LIN {X 0,Y 572.962,Z 472.956,A -85,B 0,C 180,E1 -2254.924,E2 -2254.924} C_VEL
LIN {X 0,Y 573.098,Z 467.876,A -85,B 0,C 180,E1 -2255.981,E2 -2255.981} C_VEL
LIN {X 0,Y 573.102,Z 461.481,A -85,B 0,C 180,E1 -2257.042,E2 -2257.042} C_VEL
LIN {X 0,Y 573.176,Z 453.495,A -85,B 0,C 180,E1 -2258.104,E2 -2258.104} C_VEL
LIN {X 0,Y 573.253,Z 445.356,A -85,B 0,C 180,E1 -2258.991,E2 -2258.991} C_VEL
LIN {X 0,Y 573.348,Z 435.426,A -85,B 0,C 180,E1 -2259.879,E2 -2259.879} C_VEL
LIN {X 0,Y 573.504,Z 424.221,A -85,B 0,C 180,E1 -2260.679,E2 -2260.679} C_VEL
LIN {X 0,Y 573.624,Z 413.221,A -85,B 0,C 180,E1 -2261.303,E2 -2261.303} C_VEL
LIN {X 0,Y 573.702,Z 401.041,A -85,B 0,C 180,E1 -2261.838,E2 -2261.838} C_VEL
LIN {X 0,Y 573.81,Z 388.273,A -85,B 0,C 180,E1 -2262.24,E2 -2262.24} C_VEL
LIN {X 0,Y 573.89,Z 374.763,A -85,B 0,C 180,E1 -2262.507,E2 -2262.507} C_VEL
LIN {X 0,Y 573.929,Z 274.251,A -85,B 0,C 180,E1 -2263.776,E2 -2263.776} C_VEL
LIN {X 0,Y 573.424,Z 270.457,A -85,B 0,C 180,E1 -2263.847,E2 -2263.847} C_VEL
LIN {X 0,Y 573.615,Z 247.392,A -85,B 0,C 180,E1 -2267.001,E2 -2267.001} C_VEL
LIN {X 0,Y 573.874,Z 225.362,A -85,B 0,C 180,E1 -2270.051,E2 -2270.051} C_VEL
LIN {X 0,Y 574.038,Z 204.991,A -85,B 0,C 180,E1 -2272.871,E2 -2272.871} C_VEL
LIN {X 0,Y 573.669,Z 200.428,A -85,B 0,C 180,E1 -2273.527,E2 -2273.527} C_VEL
LIN {X 0,Y 573.234,Z 198.084,A -85,B 0,C 180,E1 -2273.91,E2 -2273.91} C_VEL
LIN {X 0,Y 573.256,Z 198.078,A -85,B 0,C 180,E1 -2276.496,E2 -2276.496} C_VEL
LIN {X 0,Y 573.25,Z 198.075,A -85,B 0,C 180,E1 -2279.362,E2 -2279.362} C_VEL
LIN {X 0,Y 573.232,Z 198.082,A -85,B 0,C 180,E1 -2282.225,E2 -2282.225} C_VEL
LIN {X 0,Y 573.229,Z 198.076,A -85,B 0,C 180,E1 -2284.77,E2 -2284.77} C_VEL
LIN {X 0,Y 573.23,Z 198.076,A -85,B 0,C 180,E1 -2287.162,E2 -2287.162} C_VEL
LIN {X 0,Y 573.223,Z 198.081,A -85,B 0,C 180,E1 -2289.603,E2 -2289.603} C_VEL
LIN {X 0,Y 573.213,Z 198.078,A -85,B 0,C 180,E1 -2292.638,E2 -2292.638} C_VEL
LIN {X 0,Y 573.206,Z 198.085,A -85,B 0,C 180,E1 -2295.663,E2 -2295.663} C_VEL
LIN {X 0,Y 573.225,Z 198.076,A -85,B 0,C 180,E1 -2298.542,E2 -2298.542} C_VEL
LIN {X 0,Y 573.214,Z 198.08,A -85,B 0,C 180,E1 -2301.296,E2 -2301.296} C_VEL
LIN {X 0,Y 573.224,Z 198.081,A -85,B 0,C 180,E1 -2304.008,E2 -2304.008} C_VEL
LIN {X 0,Y 573.241,Z 198.074,A -85,B 0,C 180,E1 -2306.516,E2 -2306.516} C_VEL
LIN {X 0,Y 573.202,Z 198.081,A -85,B 0,C 180,E1 -2309.111,E2 -2309.111} C_VEL
LIN {X 0,Y 573.23,Z 198.083,A -85,B 0,C 180,E1 -2311.435,E2 -2311.435} C_VEL
LIN {X 0,Y 573.242,Z 198.079,A -85,B 0,C 180,E1 -2313.809,E2 -2313.809} C_VEL
LIN {X 0,Y 573.254,Z 198.074,A -85,B 0,C 180,E1 -2316.901,E2 -2316.901} C_VEL
LIN {X 0,Y 573.216,Z 198.079,A -85,B 0,C 180,E1 -2319.922,E2 -2319.922} C_VEL
LIN {X 0,Y 573.234,Z 198.079,A -85,B 0,C 180,E1 -2322.978,E2 -2322.978} C_VEL
LIN {X 0,Y 573.226,Z 198.078,A -85,B 0,C 180,E1 -2325.806,E2 -2325.806} C_VEL
LIN {X 0,Y 573.277,Z 198.071,A -85,B 0,C 180,E1 -2328.706,E2 -2328.706} C_VEL
LIN {X 0,Y 573.254,Z 198.077,A -85,B 0,C 180,E1 -2331.54,E2 -2331.54} C_VEL
LIN {X 0,Y 573.202,Z 198.082,A -85,B 0,C 180,E1 -2333.664,E2 -2333.664} C_VEL
LIN {X 0,Y 573.174,Z 198.084,A -85,B 0,C 180,E1 -2335.781,E2 -2335.781} C_VEL
LIN {X 0,Y 573.247,Z 198.074,A -85,B 0,C 180,E1 -2337.892,E2 -2337.892} C_VEL
LIN {X 0,Y 573.287,Z 198.072,A -85,B 0,C 180,E1 -2340.702,E2 -2340.702} C_VEL
LIN {X 0,Y 573.196,Z 198.082,A -85,B 0,C 180,E1 -2343.515,E2 -2343.515} C_VEL
LIN {X 0,Y 573.239,Z 198.075,A -85,B 0,C 180,E1 -2345.628,E2 -2345.628} C_VEL
LIN {X 0,Y 573.248,Z 198.076,A -85,B 0,C 180,E1 -2348.46,E2 -2348.46} C_VEL
LIN {X 0,Y 573.266,Z 198.074,A -85,B 0,C 180,E1 -2351.312,E2 -2351.312} C_VEL
LIN {X 0,Y 573.221,Z 198.08,A -85,B 0,C 180,E1 -2354.426,E2 -2354.426} C_VEL
LIN {X 0,Y 573.245,Z 198.078,A -85,B 0,C 180,E1 -2357.112,E2 -2357.112} C_VEL
LIN {X 0,Y 573.21,Z 198.079,A -85,B 0,C 180,E1 -2360.078,E2 -2360.078} C_VEL
LIN {X 0,Y 573.218,Z 198.08,A -85,B 0,C 180,E1 -2363.156,E2 -2363.156} C_VEL
LIN {X 0,Y 573.202,Z 198.085,A -85,B 0,C 180,E1 -2364.418,E2 -2364.418} C_VEL
LIN {X 0,Y 572.571,Z 198.169,A -85,B 0,C 180,E1 -2365.004,E2 -2365.004} C_VEL
LIN {X 0,Y 569.731,Z 198.522,A -85,B 0,C 180,E1 -2365.956,E2 -2365.956} C_VEL
LIN {X 0,Y 567.305,Z 198.822,A -85,B 0,C 180,E1 -2366.722,E2 -2366.722} C_VEL
LIN {X 0,Y 566.255,Z 198.945,A -85,B 0,C 180,E1 -2367.314,E2 -2367.314} C_VEL
LIN {X 0,Y 566.166,Z 198.955,A -85,B 0,C 180,E1 -2367.514,E2 -2367.514} C_VEL
LIN {X 0,Y 566.154,Z 198.957,A -85,B 0,C 180,E1 -2369.771,E2 -2369.771} C_VEL
LIN {X 0,Y 566.165,Z 198.964,A -85,B 0,C 180,E1 -2372.434,E2 -2372.434} C_VEL
LIN {X 0,Y 566.169,Z 198.957,A -85,B 0,C 180,E1 -2374.997,E2 -2374.997} C_VEL
LIN {X 0,Y 566.154,Z 198.957,A -85,B 0,C 180,E1 -2377.464,E2 -2377.464} C_VEL
LIN {X 0,Y 566.185,Z 198.96,A -85,B 0,C 180,E1 -2380.201,E2 -2380.201} C_VEL
LIN {X 0,Y 566.173,Z 198.955,A -85,B 0,C 180,E1 -2383.057,E2 -2383.057} C_VEL
LIN {X 0,Y 566.163,Z 198.962,A -85,B 0,C 180,E1 -2386.052,E2 -2386.052} C_VEL
LIN {X 0,Y 566.181,Z 198.955,A -85,B 0,C 180,E1 -2388.867,E2 -2388.867} C_VEL
LIN {X 0,Y 566.158,Z 198.958,A -85,B 0,C 180,E1 -2391.64,E2 -2391.64} C_VEL
LIN {X 0,Y 566.179,Z 198.961,A -85,B 0,C 180,E1 -2394.314,E2 -2394.314} C_VEL
LIN {X 0,Y 566.205,Z 198.951,A -85,B 0,C 180,E1 -2396.902,E2 -2396.902} C_VEL
LIN {X 0,Y 566.164,Z 198.957,A -85,B 0,C 180,E1 -2399.411,E2 -2399.411} C_VEL
LIN {X 0,Y 566.194,Z 198.959,A -85,B 0,C 180,E1 -2401.861,E2 -2401.861} C_VEL
LIN {X 0,Y 566.199,Z 198.956,A -85,B 0,C 180,E1 -2404.254,E2 -2404.254} C_VEL
LIN {X 0,Y 566.156,Z 198.957,A -85,B 0,C 180,E1 -2406.722,E2 -2406.722} C_VEL
LIN {X 0,Y 566.193,Z 198.958,A -85,B 0,C 180,E1 -2409.665,E2 -2409.665} C_VEL
LIN {X 0,Y 566.179,Z 198.954,A -85,B 0,C 180,E1 -2412.671,E2 -2412.671} C_VEL
LIN {X 0,Y 566.213,Z 198.957,A -85,B 0,C 180,E1 -2415.629,E2 -2415.629} C_VEL
LIN {X 0,Y 566.23,Z 198.947,A -85,B 0,C 180,E1 -2418.678,E2 -2418.678} C_VEL
LIN {X 0,Y 566.219,Z 198.954,A -85,B 0,C 180,E1 -2421.436,E2 -2421.436} C_VEL
LIN {X 0,Y 566.249,Z 198.948,A -85,B 0,C 180,E1 -2424.303,E2 -2424.303} C_VEL
LIN {X 0,Y 566.2,Z 199.072,A -85,B 0,C 180,E1 -2426.621,E2 -2426.621} C_VEL
LIN {X 0,Y 566.394,Z 207.555,A -85,B 0,C 180,E1 -2428.224,E2 -2428.224} C_VEL
LIN {X 0,Y 566.201,Z 222.6,A -85,B 0,C 180,E1 -2431.046,E2 -2431.046} C_VEL
LIN {X 0,Y 567.188,Z 228.36,A -85,B 0,C 180,E1 -2431.155,E2 -2431.155} C_VEL
LIN {X 0,Y 566.924,Z 328.742,A -85,B 0,C 180,E1 -2432.443,E2 -2432.443} C_VEL
LIN {X 0,Y 566.819,Z 341.931,A -85,B 0,C 180,E1 -2432.755,E2 -2432.755} C_VEL
LIN {X 0,Y 566.731,Z 354.545,A -85,B 0,C 180,E1 -2433.2,E2 -2433.2} C_VEL
LIN {X 0,Y 566.593,Z 365.826,A -85,B 0,C 180,E1 -2433.735,E2 -2433.735} C_VEL
LIN {X 0,Y 566.423,Z 377.466,A -85,B 0,C 180,E1 -2434.448,E2 -2434.448} C_VEL
LIN {X 0,Y 566.31,Z 387.918,A -85,B 0,C 180,E1 -2435.252,E2 -2435.252} C_VEL
LIN {X 0,Y 566.171,Z 396.509,A -85,B 0,C 180,E1 -2436.057,E2 -2436.057} C_VEL
LIN {X 0,Y 566.112,Z 404.244,A -85,B 0,C 180,E1 -2436.93,E2 -2436.93} C_VEL
LIN {X 0,Y 566.044,Z 412.234,A -85,B 0,C 180,E1 -2438.03,E2 -2438.03} C_VEL
LIN {X 0,Y 565.982,Z 417.564,A -85,B 0,C 180,E1 -2438.93,E2 -2438.93} C_VEL
LIN {X 0,Y 565.946,Z 422.761,A -85,B 0,C 180,E1 -2440.012,E2 -2440.012} C_VEL
LIN {X 0,Y 565.91,Z 426.988,A -85,B 0,C 180,E1 -2441.159,E2 -2441.159} C_VEL
LIN {X 0,Y 565.868,Z 429.791,A -85,B 0,C 180,E1 -2442.189,E2 -2442.189} C_VEL
LIN {X 0,Y 565.844,Z 431.212,A -85,B 0,C 180,E1 -2442.919,E2 -2442.919} C_VEL
LIN {X 0,Y 565.862,Z 432.216,A -85,B 0,C 180,E1 -2443.649,E2 -2443.649} C_VEL
LIN {X 0,Y 565.875,Z 432.818,A -85,B 0,C 180,E1 -2444.382,E2 -2444.382} C_VEL
LIN {X 0,Y 565.803,Z 432.99,A -85,B 0,C 180,E1 -2445.12,E2 -2445.12} C_VEL
LIN {X 0,Y 565.81,Z 432.718,A -85,B 0,C 180,E1 -2445.858,E2 -2445.858} C_VEL
LIN {X 0,Y 565.852,Z 431.495,A -85,B 0,C 180,E1 -2446.991,E2 -2446.991} C_VEL
LIN {X 0,Y 565.892,Z 428.378,A -85,B 0,C 180,E1 -2448.463,E2 -2448.463} C_VEL
LIN {X 0,Y 565.927,Z 424.709,A -85,B 0,C 180,E1 -2449.59,E2 -2449.59} C_VEL
LIN {X 0,Y 565.945,Z 419.781,A -85,B 0,C 180,E1 -2450.726,E2 -2450.726} C_VEL
LIN {X 0,Y 566.005,Z 413.426,A -85,B 0,C 180,E1 -2451.869,E2 -2451.869} C_VEL
LIN {X 0,Y 566.078,Z 405.548,A -85,B 0,C 180,E1 -2452.998,E2 -2452.998} C_VEL
LIN {X 0,Y 566.185,Z 396.971,A -85,B 0,C 180,E1 -2453.986,E2 -2453.986} C_VEL
LIN {X 0,Y 566.313,Z 386.516,A -85,B 0,C 180,E1 -2454.956,E2 -2454.956} C_VEL
LIN {X 0,Y 566.431,Z 376.094,A -85,B 0,C 180,E1 -2455.737,E2 -2455.737} C_VEL
LIN {X 0,Y 566.607,Z 364.554,A -85,B 0,C 180,E1 -2456.421,E2 -2456.421} C_VEL
LIN {X 0,Y 566.73,Z 351.798,A -85,B 0,C 180,E1 -2457.001,E2 -2457.001} C_VEL
LIN {X 0,Y 566.834,Z 339.084,A -85,B 0,C 180,E1 -2457.418,E2 -2457.418} C_VEL
LIN {X 0,Y 566.894,Z 326.866,A -85,B 0,C 180,E1 -2457.677,E2 -2457.677} C_VEL
LIN {X 0,Y 567.16,Z 228.196,A -85,B 0,C 180,E1 -2458.938,E2 -2458.938} C_VEL
LIN {X 0,Y 566.194,Z 222.551,A -85,B 0,C 180,E1 -2459.053,E2 -2459.053} C_VEL
LIN {X 0,Y 566.348,Z 207.789,A -85,B 0,C 180,E1 -2461.828,E2 -2461.828} C_VEL
LIN {X 0,Y 566.256,Z 198.949,A -85,B 0,C 180,E1 -2463.465,E2 -2463.465} C_VEL
LIN {X 0,Y 566.205,Z 198.959,A -85,B 0,C 180,E1 -2466.567,E2 -2466.567} C_VEL
LIN {X 0,Y 566.201,Z 198.953,A -85,B 0,C 180,E1 -2469.684,E2 -2469.684} C_VEL
LIN {X 0,Y 566.214,Z 198.956,A -85,B 0,C 180,E1 -2472.084,E2 -2472.084} C_VEL
LIN {X 0,Y 566.156,Z 198.958,A -85,B 0,C 180,E1 -2475.034,E2 -2475.034} C_VEL
LIN {X 0,Y 566.206,Z 198.956,A -85,B 0,C 180,E1 -2477.912,E2 -2477.912} C_VEL
LIN {X 0,Y 566.204,Z 198.953,A -85,B 0,C 180,E1 -2480.726,E2 -2480.726} C_VEL
LIN {X 0,Y 566.195,Z 198.957,A -85,B 0,C 180,E1 -2483.782,E2 -2483.782} C_VEL
LIN {X 0,Y 566.205,Z 198.956,A -85,B 0,C 180,E1 -2486.261,E2 -2486.261} C_VEL
LIN {X 0,Y 566.179,Z 198.953,A -85,B 0,C 180,E1 -2488.919,E2 -2488.919} C_VEL
LIN {X 0,Y 566.2,Z 198.959,A -85,B 0,C 180,E1 -2491.791,E2 -2491.791} C_VEL
LIN {X 0,Y 566.197,Z 198.954,A -85,B 0,C 180,E1 -2494.25,E2 -2494.25} C_VEL
LIN {X 0,Y 566.207,Z 198.95,A -85,B 0,C 180,E1 -2496.701,E2 -2496.701} C_VEL
LIN {X 0,Y 566.195,Z 198.96,A -85,B 0,C 180,E1 -2499.662,E2 -2499.662} C_VEL
LIN {X 0,Y 566.242,Z 198.946,A -85,B 0,C 180,E1 -2502.868,E2 -2502.868} C_VEL
LIN {X 0,Y 566.207,Z 198.959,A -85,B 0,C 180,E1 -2505.626,E2 -2505.626} C_VEL
LIN {X 0,Y 566.24,Z 198.946,A -85,B 0,C 180,E1 -2508.653,E2 -2508.653} C_VEL
LIN {X 0,Y 566.217,Z 198.957,A -85,B 0,C 180,E1 -2511.434,E2 -2511.434} C_VEL
LIN {X 0,Y 566.186,Z 198.959,A -85,B 0,C 180,E1 -2513.586,E2 -2513.586} C_VEL
LIN {X 0,Y 566.154,Z 198.959,A -85,B 0,C 180,E1 -2515.729,E2 -2515.729} C_VEL
LIN {X 0,Y 566.239,Z 198.948,A -85,B 0,C 180,E1 -2517.866,E2 -2517.866} C_VEL
LIN {X 0,Y 566.244,Z 198.945,A -85,B 0,C 180,E1 -2520,E2 -2520} C_VEL
LIN {X 0,Y 566.243,Z 198.949,A -85,B 0,C 180,E1 -2522.846,E2 -2522.846} C_VEL
LIN {X 0,Y 566.225,Z 198.948,A -85,B 0,C 180,E1 -2525.699,E2 -2525.699} C_VEL
LIN {X 0,Y 566.17,Z 198.957,A -85,B 0,C 180,E1 -2528.567,E2 -2528.567} C_VEL
LIN {X 0,Y 566.226,Z 198.95,A -85,B 0,C 180,E1 -2531.455,E2 -2531.455} C_VEL
LIN {X 0,Y 566.192,Z 198.954,A -85,B 0,C 180,E1 -2534.505,E2 -2534.505} C_VEL
LIN {X 0,Y 566.162,Z 198.958,A -85,B 0,C 180,E1 -2537.333,E2 -2537.333} C_VEL
LIN {X 0,Y 566.178,Z 198.956,A -85,B 0,C 180,E1 -2540.339,E2 -2540.339} C_VEL
LIN {X 0,Y 566.133,Z 198.961,A -85,B 0,C 180,E1 -2543.281,E2 -2543.281} C_VEL
LIN {X 0,Y 566.167,Z 198.955,A -85,B 0,C 180,E1 -2545.752,E2 -2545.752} C_VEL
LIN {X 0,Y 566.156,Z 198.959,A -85,B 0,C 180,E1 -2548.2,E2 -2548.2} C_VEL
LIN {X 0,Y 566.159,Z 198.958,A -85,B 0,C 180,E1 -2551.077,E2 -2551.077} C_VEL
LIN {X 0,Y 566.171,Z 198.955,A -85,B 0,C 180,E1 -2553.734,E2 -2553.734} C_VEL
LIN {X 0,Y 566.159,Z 198.964,A -85,B 0,C 180,E1 -2556.573,E2 -2556.573} C_VEL
LIN {X 0,Y 566.191,Z 198.954,A -85,B 0,C 180,E1 -2559.687,E2 -2559.687} C_VEL
LIN {X 0,Y 566.193,Z 198.956,A -85,B 0,C 180,E1 -2562.09,E2 -2562.09} C_VEL
LIN {X 0,Y 566.152,Z 198.958,A -85,B 0,C 180,E1 -2565.038,E2 -2565.038} C_VEL
LIN {X 0,Y 566.162,Z 198.961,A -85,B 0,C 180,E1 -2567.911,E2 -2567.911} C_VEL
LIN {X 0,Y 566.199,Z 198.953,A -85,B 0,C 180,E1 -2570.728,E2 -2570.728} C_VEL
LIN {X 0,Y 566.193,Z 198.957,A -85,B 0,C 180,E1 -2573.787,E2 -2573.787} C_VEL
LIN {X 0,Y 566.204,Z 198.957,A -85,B 0,C 180,E1 -2576.268,E2 -2576.268} C_VEL
LIN {X 0,Y 566.183,Z 198.954,A -85,B 0,C 180,E1 -2578.926,E2 -2578.926} C_VEL
LIN {X 0,Y 566.184,Z 198.963,A -85,B 0,C 180,E1 -2581.857,E2 -2581.857} C_VEL
LIN {X 0,Y 566.204,Z 198.957,A -85,B 0,C 180,E1 -2584.252,E2 -2584.252} C_VEL
LIN {X 0,Y 566.222,Z 199.029,A -85,B 0,C 180,E1 -2586.016,E2 -2586.016} C_VEL
LIN {X 0,Y 567.041,Z 204.539,A -85,B 0,C 180,E1 -2586.828,E2 -2586.828} C_VEL
LIN {X 0,Y 566.895,Z 223.622,A -85,B 0,C 180,E1 -2589.5,E2 -2589.5} C_VEL
LIN {X 0,Y 566.663,Z 243.988,A -85,B 0,C 180,E1 -2592.311,E2 -2592.311} C_VEL
LIN {X 0,Y 566.474,Z 265.273,A -85,B 0,C 180,E1 -2595.264,E2 -2595.264} C_VEL
LIN {X 0,Y 566.411,Z 270.522,A -85,B 0,C 180,E1 -2595.987,E2 -2595.987} C_VEL
LIN {X 0,Y 567.165,Z 277.243,A -85,B 0,C 180,E1 -2596.095,E2 -2596.095} C_VEL
LIN {X 0,Y 566.971,Z 378.942,A -85,B 0,C 180,E1 -2597.403,E2 -2597.403} C_VEL
LIN {X 0,Y 566.843,Z 392.214,A -85,B 0,C 180,E1 -2597.719,E2 -2597.719} C_VEL
LIN {X 0,Y 566.741,Z 404.374,A -85,B 0,C 180,E1 -2598.148,E2 -2598.148} C_VEL
LIN {X 0,Y 566.629,Z 416.064,A -85,B 0,C 180,E1 -2598.703,E2 -2598.703} C_VEL
LIN {X 0,Y 566.486,Z 426.902,A -85,B 0,C 180,E1 -2599.365,E2 -2599.365} C_VEL
LIN {X 0,Y 566.337,Z 437.535,A -85,B 0,C 180,E1 -2600.175,E2 -2600.175} C_VEL
LIN {X 0,Y 566.207,Z 447.109,A -85,B 0,C 180,E1 -2601.074,E2 -2601.074} C_VEL
LIN {X 0,Y 566.113,Z 454.956,A -85,B 0,C 180,E1 -2601.971,E2 -2601.971} C_VEL
LIN {X 0,Y 566.002,Z 462.619,A -85,B 0,C 180,E1 -2603.046,E2 -2603.046} C_VEL
LIN {X 0,Y 566.004,Z 469.676,A -85,B 0,C 180,E1 -2604.298,E2 -2604.298} C_VEL
LIN {X 0,Y 565.933,Z 474.369,A -85,B 0,C 180,E1 -2605.369,E2 -2605.369} C_VEL
LIN {X 0,Y 565.927,Z 477.955,A -85,B 0,C 180,E1 -2606.439,E2 -2606.439} C_VEL
LIN {X 0,Y 565.878,Z 479.805,A -85,B 0,C 180,E1 -2607.151,E2 -2607.151} C_VEL
LIN {X 0,Y 565.846,Z 482.183,A -85,B 0,C 180,E1 -2608.575,E2 -2608.575} C_VEL
LIN {X 0,Y 565.839,Z 483,A -85,B 0,C 180,E1 -2609.999,E2 -2609.999} C_VEL
LIN {X 0,Y 565.846,Z 482.187,A -85,B 0,C 180,E1 -2611.422,E2 -2611.422} C_VEL
LIN {X 0,Y 565.877,Z 479.813,A -85,B 0,C 180,E1 -2612.846,E2 -2612.846} C_VEL
LIN {X 0,Y 565.926,Z 476.9,A -85,B 0,C 180,E1 -2613.915,E2 -2613.915} C_VEL
LIN {X 0,Y 565.877,Z 472.955,A -85,B 0,C 180,E1 -2614.986,E2 -2614.986} C_VEL
LIN {X 0,Y 566.007,Z 467.876,A -85,B 0,C 180,E1 -2616.057,E2 -2616.057} C_VEL
LIN {X 0,Y 566.039,Z 461.481,A -85,B 0,C 180,E1 -2617.13,E2 -2617.13} C_VEL
LIN {X 0,Y 566.132,Z 453.494,A -85,B 0,C 180,E1 -2618.206,E2 -2618.206} C_VEL
LIN {X 0,Y 566.227,Z 445.355,A -85,B 0,C 180,E1 -2619.103,E2 -2619.103} C_VEL
LIN {X 0,Y 566.349,Z 435.425,A -85,B 0,C 180,E1 -2620.003,E2 -2620.003} C_VEL
LIN {X 0,Y 566.508,Z 424.32,A -85,B 0,C 180,E1 -2620.806,E2 -2620.806} C_VEL
LIN {X 0,Y 566.656,Z 413.219,A -85,B 0,C 180,E1 -2621.443,E2 -2621.443} C_VEL
LIN {X 0,Y 566.756,Z 401.039,A -85,B 0,C 180,E1 -2621.985,E2 -2621.985} C_VEL
LIN {X 0,Y 566.894,Z 388.272,A -85,B 0,C 180,E1 -2622.391,E2 -2622.391} C_VEL
LIN {X 0,Y 566.971,Z 374.762,A -85,B 0,C 180,E1 -2622.662,E2 -2622.662} C_VEL
LIN {X 0,Y 567.043,Z 274.921,A -85,B 0,C 180,E1 -2623.938,E2 -2623.938} C_VEL
LIN {X 0,Y 566.428,Z 270.457,A -85,B 0,C 180,E1 -2624.022,E2 -2624.022} C_VEL
LIN {X 0,Y 566.642,Z 248.047,A -85,B 0,C 180,E1 -2627.125,E2 -2627.125} C_VEL
LIN {X 0,Y 566.901,Z 226.406,A -85,B 0,C 180,E1 -2630.119,E2 -2630.119} C_VEL
LIN {X 0,Y 567.105,Z 206.052,A -85,B 0,C 180,E1 -2632.974,E2 -2632.974} C_VEL
LIN {X 0,Y 566.796,Z 202.108,A -85,B 0,C 180,E1 -2633.548,E2 -2633.548} C_VEL
LIN {X 0,Y 566.207,Z 198.96,A -85,B 0,C 180,E1 -2634.03,E2 -2634.03} C_VEL
LIN {X 0,Y 566.221,Z 198.953,A -85,B 0,C 180,E1 -2636.661,E2 -2636.661} C_VEL
LIN {X 0,Y 566.188,Z 198.958,A -85,B 0,C 180,E1 -2639.765,E2 -2639.765} C_VEL
LIN {X 0,Y 566.185,Z 198.957,A -85,B 0,C 180,E1 -2642.426,E2 -2642.426} C_VEL
LIN {X 0,Y 566.191,Z 198.952,A -85,B 0,C 180,E1 -2644.991,E2 -2644.991} C_VEL
LIN {X 0,Y 566.173,Z 198.957,A -85,B 0,C 180,E1 -2647.457,E2 -2647.457} C_VEL
LIN {X 0,Y 566.201,Z 198.956,A -85,B 0,C 180,E1 -2650.194,E2 -2650.194} C_VEL
LIN {X 0,Y 566.175,Z 198.954,A -85,B 0,C 180,E1 -2653.05,E2 -2653.05} C_VEL
LIN {X 0,Y 566.17,Z 198.961,A -85,B 0,C 180,E1 -2656.044,E2 -2656.044} C_VEL
LIN {X 0,Y 566.194,Z 198.952,A -85,B 0,C 180,E1 -2658.862,E2 -2658.862} C_VEL
LIN {X 0,Y 566.155,Z 198.965,A -85,B 0,C 180,E1 -2661.634,E2 -2661.634} C_VEL
LIN {X 0,Y 566.172,Z 198.956,A -85,B 0,C 180,E1 -2664.308,E2 -2664.308} C_VEL
LIN {X 0,Y 566.188,Z 198.953,A -85,B 0,C 180,E1 -2666.895,E2 -2666.895} C_VEL
LIN {X 0,Y 566.152,Z 198.964,A -85,B 0,C 180,E1 -2669.405,E2 -2669.405} C_VEL
LIN {X 0,Y 566.18,Z 198.958,A -85,B 0,C 180,E1 -2671.855,E2 -2671.855} C_VEL
LIN {X 0,Y 566.177,Z 198.955,A -85,B 0,C 180,E1 -2674.249,E2 -2674.249} C_VEL
LIN {X 0,Y 566.178,Z 198.962,A -85,B 0,C 180,E1 -2677.368,E2 -2677.368} C_VEL
LIN {X 0,Y 566.178,Z 198.96,A -85,B 0,C 180,E1 -2679.661,E2 -2679.661} C_VEL
LIN {X 0,Y 566.22,Z 198.951,A -85,B 0,C 180,E1 -2682.867,E2 -2682.867} C_VEL
LIN {X 0,Y 566.185,Z 198.958,A -85,B 0,C 180,E1 -2685.625,E2 -2685.625} C_VEL
LIN {X 0,Y 566.236,Z 198.948,A -85,B 0,C 180,E1 -2688.643,E2 -2688.643} C_VEL
LIN {X 0,Y 566.197,Z 198.958,A -85,B 0,C 180,E1 -2691.434,E2 -2691.434} C_VEL
LIN {X 0,Y 566.168,Z 198.959,A -85,B 0,C 180,E1 -2693.585,E2 -2693.585} C_VEL
LIN {X 0,Y 566.133,Z 198.961,A -85,B 0,C 180,E1 -2695.728,E2 -2695.728} C_VEL
LIN {X 0,Y 566.219,Z 198.949,A -85,B 0,C 180,E1 -2697.866,E2 -2697.866} C_VEL
LIN {X 0,Y 566.256,Z 198.948,A -85,B 0,C 180,E1 -2700.711,E2 -2700.711} C_VEL
LIN {X 0,Y 566.147,Z 198.96,A -85,B 0,C 180,E1 -2703.558,E2 -2703.558} C_VEL
LIN {X 0,Y 566.205,Z 198.951,A -85,B 0,C 180,E1 -2705.699,E2 -2705.699} C_VEL
LIN {X 0,Y 566.19,Z 198.956,A -85,B 0,C 180,E1 -2708.566,E2 -2708.566} C_VEL
LIN {X 0,Y 566.204,Z 198.952,A -85,B 0,C 180,E1 -2711.455,E2 -2711.455} C_VEL
LIN {X 0,Y 566.174,Z 198.959,A -85,B 0,C 180,E1 -2714.508,E2 -2714.508} C_VEL
LIN {X 0,Y 566.2,Z 198.953,A -85,B 0,C 180,E1 -2717.331,E2 -2717.331} C_VEL
LIN {X 0,Y 566.172,Z 198.958,A -85,B 0,C 180,E1 -2720.338,E2 -2720.338} C_VEL
LIN {X 0,Y 566.177,Z 198.955,A -85,B 0,C 180,E1 -2723.404,E2 -2723.404} C_VEL
LIN {X 0,Y 566.171,Z 198.955,A -85,B 0,C 180,E1 -2725.751,E2 -2725.751} C_VEL
LIN {X 0,Y 566.166,Z 198.955,A -85,B 0,C 180,E1 -2727.514,E2 -2727.514} C_VEL
LIN {X 0,Y 565.488,Z 199.044,A -85,B 0,C 180,E1 -2728.108,E2 -2728.108} C_VEL
LIN {X 0,Y 562.617,Z 199.4,A -85,B 0,C 180,E1 -2729.071,E2 -2729.071} C_VEL
LIN {X 0,Y 560.203,Z 199.7,A -85,B 0,C 180,E1 -2729.847,E2 -2729.847} C_VEL
LIN {X 0,Y 559.177,Z 199.834,A -85,B 0,C 180,E1 -2730.445,E2 -2730.445} C_VEL
LIN {X 0,Y 559.098,Z 199.837,A -85,B 0,C 180,E1 -2730.648,E2 -2730.648} C_VEL
LIN {X 0,Y 559.117,Z 199.833,A -85,B 0,C 180,E1 -2733.578,E2 -2733.578} C_VEL
LIN {X 0,Y 559.147,Z 199.84,A -85,B 0,C 180,E1 -2736.454,E2 -2736.454} C_VEL
LIN {X 0,Y 559.134,Z 199.834,A -85,B 0,C 180,E1 -2738.937,E2 -2738.937} C_VEL
LIN {X 0,Y 559.152,Z 199.831,A -85,B 0,C 180,E1 -2741.771,E2 -2741.771} C_VEL
LIN {X 0,Y 559.1,Z 199.839,A -85,B 0,C 180,E1 -2744.743,E2 -2744.743} C_VEL
LIN {X 0,Y 559.129,Z 199.832,A -85,B 0,C 180,E1 -2747.26,E2 -2747.26} C_VEL
LIN {X 0,Y 559.152,Z 199.838,A -85,B 0,C 180,E1 -2750.138,E2 -2750.138} C_VEL
LIN {X 0,Y 559.119,Z 199.834,A -85,B 0,C 180,E1 -2752.895,E2 -2752.895} C_VEL
LIN {X 0,Y 559.142,Z 199.839,A -85,B 0,C 180,E1 -2756.054,E2 -2756.054} C_VEL
LIN {X 0,Y 559.136,Z 199.831,A -85,B 0,C 180,E1 -2758.984,E2 -2758.984} C_VEL
LIN {X 0,Y 559.15,Z 199.833,A -85,B 0,C 180,E1 -2761.622,E2 -2761.622} C_VEL
LIN {X 0,Y 559.161,Z 199.829,A -85,B 0,C 180,E1 -2764.705,E2 -2764.705} C_VEL
LIN {X 0,Y 559.127,Z 199.841,A -85,B 0,C 180,E1 -2767.85,E2 -2767.85} C_VEL
LIN {X 0,Y 559.181,Z 199.827,A -85,B 0,C 180,E1 -2770.497,E2 -2770.497} C_VEL
LIN {X 0,Y 559.147,Z 199.831,A -85,B 0,C 180,E1 -2773.199,E2 -2773.199} C_VEL
LIN {X 0,Y 559.153,Z 199.832,A -85,B 0,C 180,E1 -2776.186,E2 -2776.186} C_VEL
LIN {X 0,Y 559.187,Z 199.826,A -85,B 0,C 180,E1 -2779.136,E2 -2779.136} C_VEL
LIN {X 0,Y 559.194,Z 199.829,A -85,B 0,C 180,E1 -2782.055,E2 -2782.055} C_VEL
LIN {X 0,Y 559.241,Z 199.821,A -85,B 0,C 180,E1 -2784.955,E2 -2784.955} C_VEL
LIN {X 0,Y 559.168,Z 200.002,A -85,B 0,C 180,E1 -2786.579,E2 -2786.579} C_VEL
LIN {X 0,Y 559.315,Z 206.697,A -85,B 0,C 180,E1 -2787.841,E2 -2787.841} C_VEL
LIN {X 0,Y 559.247,Z 220.051,A -85,B 0,C 180,E1 -2790.361,E2 -2790.361} C_VEL
LIN {X 0,Y 559.177,Z 222.835,A -85,B 0,C 180,E1 -2790.879,E2 -2790.879} C_VEL
LIN {X 0,Y 560.273,Z 229.137,A -85,B 0,C 180,E1 -2790.989,E2 -2790.989} C_VEL
LIN {X 0,Y 560.017,Z 329.157,A -85,B 0,C 180,E1 -2792.294,E2 -2792.294} C_VEL
LIN {X 0,Y 559.912,Z 341.452,A -85,B 0,C 180,E1 -2792.586,E2 -2792.586} C_VEL
LIN {X 0,Y 559.767,Z 354.771,A -85,B 0,C 180,E1 -2793.06,E2 -2793.06} C_VEL
LIN {X 0,Y 559.626,Z 365.992,A -85,B 0,C 180,E1 -2793.601,E2 -2793.601} C_VEL
LIN {X 0,Y 559.418,Z 377.599,A -85,B 0,C 180,E1 -2794.324,E2 -2794.324} C_VEL
LIN {X 0,Y 559.31,Z 388.021,A -85,B 0,C 180,E1 -2795.137,E2 -2795.137} C_VEL
LIN {X 0,Y 559.12,Z 396.605,A -85,B 0,C 180,E1 -2795.953,E2 -2795.953} C_VEL
LIN {X 0,Y 559.07,Z 404.696,A -85,B 0,C 180,E1 -2796.882,E2 -2796.882} C_VEL
LIN {X 0,Y 558.98,Z 412.292,A -85,B 0,C 180,E1 -2797.95,E2 -2797.95} C_VEL
LIN {X 0,Y 558.878,Z 418.546,A -85,B 0,C 180,E1 -2799.044,E2 -2799.044} C_VEL
LIN {X 0,Y 558.852,Z 423.523,A -85,B 0,C 180,E1 -2800.141,E2 -2800.141} C_VEL
LIN {X 0,Y 558.808,Z 427.228,A -85,B 0,C 180,E1 -2801.191,E2 -2801.191} C_VEL
LIN {X 0,Y 558.773,Z 430.189,A -85,B 0,C 180,E1 -2802.346,E2 -2802.346} C_VEL
LIN {X 0,Y 558.743,Z 431.513,A -85,B 0,C 180,E1 -2803.086,E2 -2803.086} C_VEL
LIN {X 0,Y 558.788,Z 432.855,A -85,B 0,C 180,E1 -2804.432,E2 -2804.432} C_VEL
LIN {X 0,Y 558.707,Z 432.947,A -85,B 0,C 180,E1 -2805.317,E2 -2805.317} C_VEL
LIN {X 0,Y 558.727,Z 432.587,A -85,B 0,C 180,E1 -2806.065,E2 -2806.065} C_VEL
LIN {X 0,Y 558.761,Z 431.398,A -85,B 0,C 180,E1 -2807.077,E2 -2807.077} C_VEL
LIN {X 0,Y 558.777,Z 428.832,A -85,B 0,C 180,E1 -2808.326,E2 -2808.326} C_VEL
LIN {X 0,Y 558.827,Z 425.582,A -85,B 0,C 180,E1 -2809.4,E2 -2809.4} C_VEL
LIN {X 0,Y 558.842,Z 420.654,A -85,B 0,C 180,E1 -2810.617,E2 -2810.617} C_VEL
LIN {X 0,Y 558.915,Z 414.713,A -85,B 0,C 180,E1 -2811.747,E2 -2811.747} C_VEL
LIN {X 0,Y 559.001,Z 406.755,A -85,B 0,C 180,E1 -2812.938,E2 -2812.938} C_VEL
LIN {X 0,Y 559.135,Z 398.691,A -85,B 0,C 180,E1 -2813.913,E2 -2813.913} C_VEL
LIN {X 0,Y 559.284,Z 388.71,A -85,B 0,C 180,E1 -2814.894,E2 -2814.894} C_VEL
LIN {X 0,Y 559.407,Z 377.344,A -85,B 0,C 180,E1 -2815.784,E2 -2815.784} C_VEL
LIN {X 0,Y 559.641,Z 366.253,A -85,B 0,C 180,E1 -2816.474,E2 -2816.474} C_VEL
LIN {X 0,Y 559.781,Z 354.713,A -85,B 0,C 180,E1 -2817.033,E2 -2817.033} C_VEL
LIN {X 0,Y 559.866,Z 341.394,A -85,B 0,C 180,E1 -2817.507,E2 -2817.507} C_VEL
LIN {X 0,Y 559.939,Z 329.219,A -85,B 0,C 180,E1 -2817.797,E2 -2817.797} C_VEL
LIN {X 0,Y 560.239,Z 228.963,A -85,B 0,C 180,E1 -2819.104,E2 -2819.104} C_VEL
LIN {X 0,Y 559.165,Z 222.683,A -85,B 0,C 180,E1 -2819.222,E2 -2819.222} C_VEL
LIN {X 0,Y 559.312,Z 210.352,A -85,B 0,C 180,E1 -2821.541,E2 -2821.541} C_VEL
LIN {X 0,Y 559.308,Z 200.615,A -85,B 0,C 180,E1 -2823.347,E2 -2823.347} C_VEL
LIN {X 0,Y 559.219,Z 199.826,A -85,B 0,C 180,E1 -2823.515,E2 -2823.515} C_VEL
LIN {X 0,Y 559.179,Z 199.835,A -85,B 0,C 180,E1 -2826.45,E2 -2826.45} C_VEL
LIN {X 0,Y 559.166,Z 199.831,A -85,B 0,C 180,E1 -2828.932,E2 -2828.932} C_VEL
LIN {X 0,Y 559.187,Z 199.827,A -85,B 0,C 180,E1 -2831.765,E2 -2831.765} C_VEL
LIN {X 0,Y 559.123,Z 199.836,A -85,B 0,C 180,E1 -2834.737,E2 -2834.737} C_VEL
LIN {X 0,Y 559.153,Z 199.83,A -85,B 0,C 180,E1 -2837.256,E2 -2837.256} C_VEL
LIN {X 0,Y 559.167,Z 199.836,A -85,B 0,C 180,E1 -2840.134,E2 -2840.134} C_VEL
LIN {X 0,Y 559.125,Z 199.833,A -85,B 0,C 180,E1 -2842.891,E2 -2842.891} C_VEL
LIN {X 0,Y 559.139,Z 199.833,A -85,B 0,C 180,E1 -2845.555,E2 -2845.555} C_VEL
LIN {X 0,Y 559.149,Z 199.836,A -85,B 0,C 180,E1 -2848.136,E2 -2848.136} C_VEL
LIN {X 0,Y 559.135,Z 199.831,A -85,B 0,C 180,E1 -2850.646,E2 -2850.646} C_VEL
LIN {X 0,Y 559.155,Z 199.83,A -85,B 0,C 180,E1 -2853.168,E2 -2853.168} C_VEL
LIN {X 0,Y 559.138,Z 199.835,A -85,B 0,C 180,E1 -2855.494,E2 -2855.494} C_VEL
LIN {X 0,Y 559.135,Z 199.831,A -85,B 0,C 180,E1 -2858.446,E2 -2858.446} C_VEL
LIN {X 0,Y 559.144,Z 199.831,A -85,B 0,C 180,E1 -2860.926,E2 -2860.926} C_VEL
LIN {X 0,Y 559.181,Z 199.828,A -85,B 0,C 180,E1 -2863.198,E2 -2863.198} C_VEL
LIN {X 0,Y 559.147,Z 199.831,A -85,B 0,C 180,E1 -2866.184,E2 -2866.184} C_VEL
LIN {X 0,Y 559.181,Z 199.829,A -85,B 0,C 180,E1 -2869.133,E2 -2869.133} C_VEL
LIN {X 0,Y 559.179,Z 199.826,A -85,B 0,C 180,E1 -2872.053,E2 -2872.053} C_VEL
LIN {X 0,Y 559.232,Z 199.822,A -85,B 0,C 180,E1 -2874.953,E2 -2874.953} C_VEL
LIN {X 0,Y 559.212,Z 199.823,A -85,B 0,C 180,E1 -2877.839,E2 -2877.839} C_VEL
LIN {X 0,Y 559.215,Z 199.82,A -85,B 0,C 180,E1 -2880,E2 -2880} C_VEL
LIN {X 0,Y 559.21,Z 199.825,A -85,B 0,C 180,E1 -2882.882,E2 -2882.882} C_VEL
LIN {X 0,Y 559.193,Z 199.823,A -85,B 0,C 180,E1 -2885.771,E2 -2885.771} C_VEL
LIN {X 0,Y 559.135,Z 199.834,A -85,B 0,C 180,E1 -2888.675,E2 -2888.675} C_VEL
LIN {X 0,Y 559.178,Z 199.827,A -85,B 0,C 180,E1 -2891.601,E2 -2891.601} C_VEL
LIN {X 0,Y 559.166,Z 199.831,A -85,B 0,C 180,E1 -2894.597,E2 -2894.597} C_VEL
LIN {X 0,Y 559.106,Z 199.835,A -85,B 0,C 180,E1 -2897.559,E2 -2897.559} C_VEL
LIN {X 0,Y 559.134,Z 199.831,A -85,B 0,C 180,E1 -2899.839,E2 -2899.839} C_VEL
LIN {X 0,Y 559.107,Z 199.836,A -85,B 0,C 180,E1 -2902.154,E2 -2902.154} C_VEL
LIN {X 0,Y 559.109,Z 199.838,A -85,B 0,C 180,E1 -2905.18,E2 -2905.18} C_VEL
LIN {X 0,Y 559.099,Z 199.835,A -85,B 0,C 180,E1 -2907.717,E2 -2907.717} C_VEL
LIN {X 0,Y 559.12,Z 199.837,A -85,B 0,C 180,E1 -2910.185,E2 -2910.185} C_VEL
LIN {X 0,Y 559.126,Z 199.839,A -85,B 0,C 180,E1 -2912.717,E2 -2912.717} C_VEL
LIN {X 0,Y 559.099,Z 199.836,A -85,B 0,C 180,E1 -2915.326,E2 -2915.326} C_VEL
LIN {X 0,Y 559.106,Z 199.838,A -85,B 0,C 180,E1 -2918.02,E2 -2918.02} C_VEL
LIN {X 0,Y 559.138,Z 199.832,A -85,B 0,C 180,E1 -2920.814,E2 -2920.814} C_VEL
LIN {X 0,Y 559.128,Z 199.832,A -85,B 0,C 180,E1 -2923.198,E2 -2923.198} C_VEL
LIN {X 0,Y 559.12,Z 199.843,A -85,B 0,C 180,E1 -2926.267,E2 -2926.267} C_VEL
LIN {X 0,Y 559.141,Z 199.831,A -85,B 0,C 180,E1 -2929.189,E2 -2929.189} C_VEL
LIN {X 0,Y 559.119,Z 199.842,A -85,B 0,C 180,E1 -2931.984,E2 -2931.984} C_VEL
LIN {X 0,Y 559.136,Z 199.833,A -85,B 0,C 180,E1 -2934.787,E2 -2934.787} C_VEL
LIN {X 0,Y 559.148,Z 199.832,A -85,B 0,C 180,E1 -2937.366,E2 -2937.366} C_VEL
LIN {X 0,Y 559.142,Z 199.838,A -85,B 0,C 180,E1 -2940.144,E2 -2940.144} C_VEL
LIN {X 0,Y 559.159,Z 199.831,A -85,B 0,C 180,E1 -2943.176,E2 -2943.176} C_VEL
LIN {X 0,Y 559.191,Z 200.023,A -85,B 0,C 180,E1 -2945.893,E2 -2945.893} C_VEL
LIN {X 0,Y 560.099,Z 205.652,A -85,B 0,C 180,E1 -2946.735,E2 -2946.735} C_VEL
LIN {X 0,Y 559.909,Z 224.626,A -85,B 0,C 180,E1 -2949.424,E2 -2949.424} C_VEL
LIN {X 0,Y 559.636,Z 244.992,A -85,B 0,C 180,E1 -2952.27,E2 -2952.27} C_VEL
LIN {X 0,Y 559.459,Z 265.287,A -85,B 0,C 180,E1 -2955.077,E2 -2955.077} C_VEL
LIN {X 0,Y 559.429,Z 270.522,A -85,B 0,C 180,E1 -2955.808,E2 -2955.808} C_VEL
LIN {X 0,Y 560.301,Z 278.3,A -85,B 0,C 180,E1 -2955.935,E2 -2955.935} C_VEL
LIN {X 0,Y 560.035,Z 378.942,A -85,B 0,C 180,E1 -2957.245,E2 -2957.245} C_VEL
LIN {X 0,Y 559.898,Z 392.213,A -85,B 0,C 180,E1 -2957.564,E2 -2957.564} C_VEL
LIN {X 0,Y 559.8,Z 404.373,A -85,B 0,C 180,E1 -2957.999,E2 -2957.999} C_VEL
LIN {X 0,Y 559.669,Z 415.807,A -85,B 0,C 180,E1 -2958.547,E2 -2958.547} C_VEL
LIN {X 0,Y 559.51,Z 426.9,A -85,B 0,C 180,E1 -2959.231,E2 -2959.231} C_VEL
LIN {X 0,Y 559.317,Z 437.533,A -85,B 0,C 180,E1 -2960.051,E2 -2960.051} C_VEL
LIN {X 0,Y 559.162,Z 447.109,A -85,B 0,C 180,E1 -2960.96,E2 -2960.96} C_VEL
LIN {X 0,Y 559.05,Z 454.956,A -85,B 0,C 180,E1 -2961.869,E2 -2961.869} C_VEL
LIN {X 0,Y 558.944,Z 462.619,A -85,B 0,C 180,E1 -2962.958,E2 -2962.958} C_VEL
LIN {X 0,Y 558.936,Z 469.676,A -85,B 0,C 180,E1 -2964.226,E2 -2964.226} C_VEL
LIN {X 0,Y 558.827,Z 474.37,A -85,B 0,C 180,E1 -2965.31,E2 -2965.31} C_VEL
LIN {X 0,Y 558.836,Z 477.956,A -85,B 0,C 180,E1 -2966.394,E2 -2966.394} C_VEL
LIN {X 0,Y 558.799,Z 479.805,A -85,B 0,C 180,E1 -2967.115,E2 -2967.115} C_VEL
LIN {X 0,Y 558.745,Z 482.182,A -85,B 0,C 180,E1 -2968.557,E2 -2968.557} C_VEL
LIN {X 0,Y 558.74,Z 483,A -85,B 0,C 180,E1 -2969.999,E2 -2969.999} C_VEL
LIN {X 0,Y 558.745,Z 482.186,A -85,B 0,C 180,E1 -2971.44,E2 -2971.44} C_VEL
LIN {X 0,Y 558.799,Z 479.813,A -85,B 0,C 180,E1 -2972.882,E2 -2972.882} C_VEL
LIN {X 0,Y 558.844,Z 476.9,A -85,B 0,C 180,E1 -2973.965,E2 -2973.965} C_VEL
LIN {X 0,Y 558.798,Z 472.955,A -85,B 0,C 180,E1 -2975.049,E2 -2975.049} C_VEL
LIN {X 0,Y 558.921,Z 467.877,A -85,B 0,C 180,E1 -2976.134,E2 -2976.134} C_VEL
LIN {X 0,Y 558.975,Z 461.48,A -85,B 0,C 180,E1 -2977.221,E2 -2977.221} C_VEL
LIN {X 0,Y 559.097,Z 453.494,A -85,B 0,C 180,E1 -2978.31,E2 -2978.31} C_VEL
LIN {X 0,Y 559.183,Z 445.354,A -85,B 0,C 180,E1 -2979.219,E2 -2979.219} C_VEL
LIN {X 0,Y 559.36,Z 435.424,A -85,B 0,C 180,E1 -2980.129,E2 -2980.129} C_VEL
LIN {X 0,Y 559.51,Z 424.398,A -85,B 0,C 180,E1 -2980.938,E2 -2980.938} C_VEL
LIN {X 0,Y 559.699,Z 412.184,A -85,B 0,C 180,E1 -2981.641,E2 -2981.641} C_VEL
LIN {X 0,Y 559.827,Z 399.835,A -85,B 0,C 180,E1 -2982.182,E2 -2982.182} C_VEL
LIN {X 0,Y 559.987,Z 387.356,A -85,B 0,C 180,E1 -2982.57,E2 -2982.57} C_VEL
LIN {X 0,Y 560.055,Z 374.761,A -85,B 0,C 180,E1 -2982.821,E2 -2982.821} C_VEL
LIN {X 0,Y 560.202,Z 275.926,A -85,B 0,C 180,E1 -2984.098,E2 -2984.098} C_VEL
LIN {X 0,Y 559.407,Z 270.457,A -85,B 0,C 180,E1 -2984.201,E2 -2984.201} C_VEL
LIN {X 0,Y 559.668,Z 247.569,A -85,B 0,C 180,E1 -2987.375,E2 -2987.375} C_VEL
LIN {X 0,Y 559.944,Z 224.737,A -85,B 0,C 180,E1 -2990.572,E2 -2990.572} C_VEL
LIN {X 0,Y 560.156,Z 205.862,A -85,B 0,C 180,E1 -2993.261,E2 -2993.261} C_VEL
LIN {X 0,Y 559.168,Z 199.837,A -85,B 0,C 180,E1 -2994.204,E2 -2994.204} C_VEL
LIN {X 0,Y 559.166,Z 199.83,A -85,B 0,C 180,E1 -2996.898,E2 -2996.898} C_VEL
LIN {X 0,Y 559.135,Z 199.839,A -85,B 0,C 180,E1 -2999.854,E2 -2999.854} C_VEL
LIN {X 0,Y 559.156,Z 199.83,A -85,B 0,C 180,E1 -3002.71,E2 -3002.71} C_VEL
LIN {X 0,Y 559.136,Z 199.832,A -85,B 0,C 180,E1 -3005.318,E2 -3005.318} C_VEL
LIN {X 0,Y 559.111,Z 199.843,A -85,B 0,C 180,E1 -3008.014,E2 -3008.014} C_VEL
LIN {X 0,Y 559.15,Z 199.829,A -85,B 0,C 180,E1 -3010.807,E2 -3010.807} C_VEL
LIN {X 0,Y 559.132,Z 199.839,A -85,B 0,C 180,E1 -3013.728,E2 -3013.728} C_VEL
LIN {X 0,Y 559.141,Z 199.83,A -85,B 0,C 180,E1 -3016.797,E2 -3016.797} C_VEL
LIN {X 0,Y 559.164,Z 199.829,A -85,B 0,C 180,E1 -3019.188,E2 -3019.188} C_VEL
LIN {X 0,Y 559.099,Z 199.841,A -85,B 0,C 180,E1 -3021.979,E2 -3021.979} C_VEL
LIN {X 0,Y 559.118,Z 199.833,A -85,B 0,C 180,E1 -3024.675,E2 -3024.675} C_VEL
LIN {X 0,Y 559.135,Z 199.837,A -85,B 0,C 180,E1 -3027.357,E2 -3027.357} C_VEL
LIN {X 0,Y 559.147,Z 199.832,A -85,B 0,C 180,E1 -3030.131,E2 -3030.131} C_VEL
LIN {X 0,Y 559.133,Z 199.835,A -85,B 0,C 180,E1 -3033.096,E2 -3033.096} C_VEL
LIN {X 0,Y 559.118,Z 199.843,A -85,B 0,C 180,E1 -3035.493,E2 -3035.493} C_VEL
LIN {X 0,Y 559.118,Z 199.837,A -85,B 0,C 180,E1 -3037.846,E2 -3037.846} C_VEL
LIN {X 0,Y 559.145,Z 199.83,A -85,B 0,C 180,E1 -3040.49,E2 -3040.49} C_VEL
LIN {X 0,Y 559.159,Z 199.835,A -85,B 0,C 180,E1 -3043.197,E2 -3043.197} C_VEL
LIN {X 0,Y 559.132,Z 199.832,A -85,B 0,C 180,E1 -3046.183,E2 -3046.183} C_VEL
LIN {X 0,Y 559.201,Z 199.831,A -85,B 0,C 180,E1 -3049.133,E2 -3049.133} C_VEL
LIN {X 0,Y 559.157,Z 199.829,A -85,B 0,C 180,E1 -3052.053,E2 -3052.053} C_VEL
LIN {X 0,Y 559.211,Z 199.828,A -85,B 0,C 180,E1 -3054.953,E2 -3054.953} C_VEL
LIN {X 0,Y 559.191,Z 199.825,A -85,B 0,C 180,E1 -3057.839,E2 -3057.839} C_VEL
LIN {X 0,Y 559.225,Z 199.824,A -85,B 0,C 180,E1 -3060.72,E2 -3060.72} C_VEL
LIN {X 0,Y 559.193,Z 199.831,A -85,B 0,C 180,E1 -3062.881,E2 -3062.881} C_VEL
LIN {X 0,Y 559.173,Z 199.827,A -85,B 0,C 180,E1 -3065.771,E2 -3065.771} C_VEL
LIN {X 0,Y 559.145,Z 199.835,A -85,B 0,C 180,E1 -3068.675,E2 -3068.675} C_VEL
LIN {X 0,Y 559.156,Z 199.829,A -85,B 0,C 180,E1 -3071.601,E2 -3071.601} C_VEL
LIN {X 0,Y 559.141,Z 199.836,A -85,B 0,C 180,E1 -3074.597,E2 -3074.597} C_VEL
LIN {X 0,Y 559.155,Z 199.829,A -85,B 0,C 180,E1 -3077.557,E2 -3077.557} C_VEL
LIN {X 0,Y 559.136,Z 199.839,A -85,B 0,C 180,E1 -3080.606,E2 -3080.606} C_VEL
LIN {X 0,Y 559.113,Z 199.834,A -85,B 0,C 180,E1 -3083.718,E2 -3083.718} C_VEL
LIN {X 0,Y 559.146,Z 199.832,A -85,B 0,C 180,E1 -3086.099,E2 -3086.099} C_VEL
LIN {X 0,Y 559.125,Z 199.841,A -85,B 0,C 180,E1 -3088.532,E2 -3088.532} C_VEL
LIN {X 0,Y 559.098,Z 199.837,A -85,B 0,C 180,E1 -3090.648,E2 -3090.648} C_VEL
LIN {X 0,Y 558.441,Z 199.921,A -85,B 0,C 180,E1 -3091.25,E2 -3091.25} C_VEL
LIN {X 0,Y 555.578,Z 200.279,A -85,B 0,C 180,E1 -3092.226,E2 -3092.226} C_VEL
LIN {X 0,Y 553.164,Z 200.577,A -85,B 0,C 180,E1 -3093.012,E2 -3093.012} C_VEL
LIN {X 0,Y 552.144,Z 200.702,A -85,B 0,C 180,E1 -3093.618,E2 -3093.618} C_VEL
LIN {X 0,Y 552.07,Z 200.712,A -85,B 0,C 180,E1 -3093.824,E2 -3093.824} C_VEL
LIN {X 0,Y 552.075,Z 200.715,A -85,B 0,C 180,E1 -3096.749,E2 -3096.749} C_VEL
LIN {X 0,Y 552.091,Z 200.709,A -85,B 0,C 180,E1 -3099.53,E2 -3099.53} C_VEL
LIN {X 0,Y 552.095,Z 200.717,A -85,B 0,C 180,E1 -3102.429,E2 -3102.429} C_VEL
LIN {X 0,Y 552.06,Z 200.713,A -85,B 0,C 180,E1 -3105.566,E2 -3105.566} C_VEL
LIN {X 0,Y 552.109,Z 200.71,A -85,B 0,C 180,E1 -3108.68,E2 -3108.68} C_VEL
LIN {X 0,Y 552.09,Z 200.709,A -85,B 0,C 180,E1 -3111.415,E2 -3111.415} C_VEL
LIN {X 0,Y 552.083,Z 200.719,A -85,B 0,C 180,E1 -3114.161,E2 -3114.161} C_VEL
LIN {X 0,Y 552.094,Z 200.709,A -85,B 0,C 180,E1 -3116.818,E2 -3116.818} C_VEL
LIN {X 0,Y 552.084,Z 200.711,A -85,B 0,C 180,E1 -3119.394,E2 -3119.394} C_VEL
LIN {X 0,Y 552.089,Z 200.717,A -85,B 0,C 180,E1 -3121.905,E2 -3121.905} C_VEL
LIN {X 0,Y 552.141,Z 200.703,A -85,B 0,C 180,E1 -3124.653,E2 -3124.653} C_VEL
LIN {X 0,Y 552.078,Z 200.714,A -85,B 0,C 180,E1 -3127.552,E2 -3127.552} C_VEL
LIN {X 0,Y 552.133,Z 200.706,A -85,B 0,C 180,E1 -3130.378,E2 -3130.378} C_VEL
LIN {X 0,Y 552.108,Z 200.707,A -85,B 0,C 180,E1 -3132.979,E2 -3132.979} C_VEL
LIN {X 0,Y 552.121,Z 200.711,A -85,B 0,C 180,E1 -3136.007,E2 -3136.007} C_VEL
LIN {X 0,Y 552.156,Z 200.701,A -85,B 0,C 180,E1 -3138.996,E2 -3138.996} C_VEL
LIN {X 0,Y 552.149,Z 200.708,A -85,B 0,C 180,E1 -3141.953,E2 -3141.953} C_VEL
LIN {X 0,Y 552.217,Z 200.696,A -85,B 0,C 180,E1 -3144.891,E2 -3144.891} C_VEL
LIN {X 0,Y 552.097,Z 200.785,A -85,B 0,C 180,E1 -3146.489,E2 -3146.489} C_VEL
LIN {X 0,Y 552.353,Z 205.836,A -85,B 0,C 180,E1 -3147.449,E2 -3147.449} C_VEL
LIN {X 0,Y 552.217,Z 221.267,A -85,B 0,C 180,E1 -3150.366,E2 -3150.366} C_VEL
LIN {X 0,Y 552.197,Z 223.154,A -85,B 0,C 180,E1 -3150.696,E2 -3150.696} C_VEL
LIN {X 0,Y 553.469,Z 231.668,A -85,B 0,C 180,E1 -3150.842,E2 -3150.842} C_VEL
LIN {X 0,Y 553.103,Z 329.792,A -85,B 0,C 180,E1 -3152.14,E2 -3152.14} C_VEL
LIN {X 0,Y 552.973,Z 341.953,A -85,B 0,C 180,E1 -3152.437,E2 -3152.437} C_VEL
LIN {X 0,Y 552.82,Z 355.165,A -85,B 0,C 180,E1 -3152.916,E2 -3152.916} C_VEL
LIN {X 0,Y 552.672,Z 366.29,A -85,B 0,C 180,E1 -3153.464,E2 -3153.464} C_VEL
LIN {X 0,Y 552.43,Z 377.823,A -85,B 0,C 180,E1 -3154.196,E2 -3154.196} C_VEL
LIN {X 0,Y 552.291,Z 388.174,A -85,B 0,C 180,E1 -3155.02,E2 -3155.02} C_VEL
LIN {X 0,Y 552.072,Z 396.701,A -85,B 0,C 180,E1 -3155.846,E2 -3155.846} C_VEL
LIN {X 0,Y 552.003,Z 404.442,A -85,B 0,C 180,E1 -3156.745,E2 -3156.745} C_VEL
LIN {X 0,Y 551.918,Z 412.35,A -85,B 0,C 180,E1 -3157.868,E2 -3157.868} C_VEL
LIN {X 0,Y 551.789,Z 419.504,A -85,B 0,C 180,E1 -3159.161,E2 -3159.161} C_VEL
LIN {X 0,Y 551.745,Z 424.282,A -85,B 0,C 180,E1 -3160.273,E2 -3160.273} C_VEL
LIN {X 0,Y 551.724,Z 427.494,A -85,B 0,C 180,E1 -3161.233,E2 -3161.233} C_VEL
LIN {X 0,Y 551.66,Z 430.578,A -85,B 0,C 180,E1 -3162.508,E2 -3162.508} C_VEL
LIN {X 0,Y 551.656,Z 431.811,A -85,B 0,C 180,E1 -3163.257,E2 -3163.257} C_VEL
LIN {X 0,Y 551.692,Z 432.886,A -85,B 0,C 180,E1 -3164.497,E2 -3164.497} C_VEL
LIN {X 0,Y 551.604,Z 432.903,A -85,B 0,C 180,E1 -3165.519,E2 -3165.519} C_VEL
LIN {X 0,Y 551.631,Z 432.431,A -85,B 0,C 180,E1 -3166.277,E2 -3166.277} C_VEL
LIN {X 0,Y 551.678,Z 431.297,A -85,B 0,C 180,E1 -3167.168,E2 -3167.168} C_VEL
LIN {X 0,Y 551.688,Z 428.324,A -85,B 0,C 180,E1 -3168.57,E2 -3168.57} C_VEL
LIN {X 0,Y 551.772,Z 424.466,A -85,B 0,C 180,E1 -3169.77,E2 -3169.77} C_VEL
LIN {X 0,Y 551.799,Z 419.684,A -85,B 0,C 180,E1 -3170.892,E2 -3170.892} C_VEL
LIN {X 0,Y 551.874,Z 413.302,A -85,B 0,C 180,E1 -3172.065,E2 -3172.065} C_VEL
LIN {X 0,Y 551.976,Z 405.222,A -85,B 0,C 180,E1 -3173.247,E2 -3173.247} C_VEL
LIN {X 0,Y 552.113,Z 396.767,A -85,B 0,C 180,E1 -3174.236,E2 -3174.236} C_VEL
LIN {X 0,Y 552.286,Z 387.179,A -85,B 0,C 180,E1 -3175.157,E2 -3175.157} C_VEL
LIN {X 0,Y 552.468,Z 375.909,A -85,B 0,C 180,E1 -3176.031,E2 -3176.031} C_VEL
LIN {X 0,Y 552.714,Z 364.444,A -85,B 0,C 180,E1 -3176.725,E2 -3176.725} C_VEL
LIN {X 0,Y 552.852,Z 352.486,A -85,B 0,C 180,E1 -3177.285,E2 -3177.285} C_VEL
LIN {X 0,Y 552.978,Z 339.974,A -85,B 0,C 180,E1 -3177.714,E2 -3177.714} C_VEL
LIN {X 0,Y 553.059,Z 327.464,A -85,B 0,C 180,E1 -3177.993,E2 -3177.993} C_VEL
LIN {X 0,Y 553.314,Z 229.511,A -85,B 0,C 180,E1 -3179.28,E2 -3179.28} C_VEL
LIN {X 0,Y 552.186,Z 222.819,A -85,B 0,C 180,E1 -3179.418,E2 -3179.418} C_VEL
LIN {X 0,Y 552.297,Z 213.227,A -85,B 0,C 180,E1 -3181.233,E2 -3181.233} C_VEL
LIN {X 0,Y 552.306,Z 201.592,A -85,B 0,C 180,E1 -3183.389,E2 -3183.389} C_VEL
LIN {X 0,Y 552.207,Z 200.7,A -85,B 0,C 180,E1 -3183.56,E2 -3183.56} C_VEL
LIN {X 0,Y 552.106,Z 200.713,A -85,B 0,C 180,E1 -3186.745,E2 -3186.745} C_VEL
LIN {X 0,Y 552.122,Z 200.707,A -85,B 0,C 180,E1 -3189.525,E2 -3189.525} C_VEL
LIN {X 0,Y 552.157,Z 200.701,A -85,B 0,C 180,E1 -3191.44,E2 -3191.44} C_VEL
LIN {X 0,Y 552.079,Z 200.717,A -85,B 0,C 180,E1 -3194.53,E2 -3194.53} C_VEL
LIN {X 0,Y 552.113,Z 200.708,A -85,B 0,C 180,E1 -3197.583,E2 -3197.583} C_VEL
LIN {X 0,Y 552.115,Z 200.711,A -85,B 0,C 180,E1 -3200.472,E2 -3200.472} C_VEL
LIN {X 0,Y 552.092,Z 200.709,A -85,B 0,C 180,E1 -3203.314,E2 -3203.314} C_VEL
LIN {X 0,Y 552.117,Z 200.713,A -85,B 0,C 180,E1 -3205.939,E2 -3205.939} C_VEL
LIN {X 0,Y 552.092,Z 200.71,A -85,B 0,C 180,E1 -3208.539,E2 -3208.539} C_VEL
LIN {X 0,Y 552.107,Z 200.709,A -85,B 0,C 180,E1 -3211.434,E2 -3211.434} C_VEL
LIN {X 0,Y 552.108,Z 200.707,A -85,B 0,C 180,E1 -3214.355,E2 -3214.355} C_VEL
LIN {X 0,Y 552.117,Z 200.705,A -85,B 0,C 180,E1 -3216.759,E2 -3216.759} C_VEL
LIN {X 0,Y 552.099,Z 200.708,A -85,B 0,C 180,E1 -3219.119,E2 -3219.119} C_VEL
LIN {X 0,Y 552.106,Z 200.713,A -85,B 0,C 180,E1 -3221.444,E2 -3221.444} C_VEL
LIN {X 0,Y 552.105,Z 200.715,A -85,B 0,C 180,E1 -3223.737,E2 -3223.737} C_VEL
LIN {X 0,Y 552.108,Z 200.709,A -85,B 0,C 180,E1 -3226.004,E2 -3226.004} C_VEL
LIN {X 0,Y 552.147,Z 200.704,A -85,B 0,C 180,E1 -3228.993,E2 -3228.993} C_VEL
LIN {X 0,Y 552.132,Z 200.704,A -85,B 0,C 180,E1 -3231.951,E2 -3231.951} C_VEL
LIN {X 0,Y 552.169,Z 200.699,A -85,B 0,C 180,E1 -3234.156,E2 -3234.156} C_VEL
LIN {X 0,Y 552.18,Z 200.701,A -85,B 0,C 180,E1 -3237.082,E2 -3237.082} C_VEL
LIN {X 0,Y 552.186,Z 200.696,A -85,B 0,C 180,E1 -3240,E2 -3240} C_VEL
LIN {X 0,Y 552.176,Z 200.702,A -85,B 0,C 180,E1 -3242.918,E2 -3242.918} C_VEL
LIN {X 0,Y 552.162,Z 200.698,A -85,B 0,C 180,E1 -3245.845,E2 -3245.845} C_VEL
LIN {X 0,Y 552.112,Z 200.711,A -85,B 0,C 180,E1 -3248.787,E2 -3248.787} C_VEL
LIN {X 0,Y 552.132,Z 200.703,A -85,B 0,C 180,E1 -3251.751,E2 -3251.751} C_VEL
LIN {X 0,Y 552.102,Z 200.713,A -85,B 0,C 180,E1 -3254.75,E2 -3254.75} C_VEL
LIN {X 0,Y 552.064,Z 200.712,A -85,B 0,C 180,E1 -3257.79,E2 -3257.79} C_VEL
LIN {X 0,Y 552.096,Z 200.708,A -85,B 0,C 180,E1 -3260.103,E2 -3260.103} C_VEL
LIN {X 0,Y 552.058,Z 200.718,A -85,B 0,C 180,E1 -3262.453,E2 -3262.453} C_VEL
LIN {X 0,Y 552.054,Z 200.715,A -85,B 0,C 180,E1 -3265.336,E2 -3265.336} C_VEL
LIN {X 0,Y 552.064,Z 200.713,A -85,B 0,C 180,E1 -3267.277,E2 -3267.277} C_VEL
LIN {X 0,Y 552.085,Z 200.712,A -85,B 0,C 180,E1 -3270.051,E2 -3270.051} C_VEL
LIN {X 0,Y 552.085,Z 200.714,A -85,B 0,C 180,E1 -3272.847,E2 -3272.847} C_VEL
LIN {X 0,Y 552.046,Z 200.715,A -85,B 0,C 180,E1 -3275.44,E2 -3275.44} C_VEL
LIN {X 0,Y 552.07,Z 200.713,A -85,B 0,C 180,E1 -3277.887,E2 -3277.887} C_VEL
LIN {X 0,Y 552.089,Z 200.714,A -85,B 0,C 180,E1 -3280.483,E2 -3280.483} C_VEL
LIN {X 0,Y 552.091,Z 200.709,A -85,B 0,C 180,E1 -3283.426,E2 -3283.426} C_VEL
LIN {X 0,Y 552.093,Z 200.713,A -85,B 0,C 180,E1 -3286.578,E2 -3286.578} C_VEL
LIN {X 0,Y 552.095,Z 200.71,A -85,B 0,C 180,E1 -3289.52,E2 -3289.52} C_VEL
LIN {X 0,Y 552.08,Z 200.715,A -85,B 0,C 180,E1 -3292.338,E2 -3292.338} C_VEL
LIN {X 0,Y 552.085,Z 200.711,A -85,B 0,C 180,E1 -3295.053,E2 -3295.053} C_VEL
LIN {X 0,Y 552.108,Z 200.713,A -85,B 0,C 180,E1 -3297.683,E2 -3297.683} C_VEL
LIN {X 0,Y 552.105,Z 200.713,A -85,B 0,C 180,E1 -3300.236,E2 -3300.236} C_VEL
LIN {X 0,Y 552.126,Z 200.707,A -85,B 0,C 180,E1 -3303.003,E2 -3303.003} C_VEL
LIN {X 0,Y 552.132,Z 200.846,A -85,B 0,C 180,E1 -3305.739,E2 -3305.739} C_VEL
LIN {X 0,Y 553.203,Z 207.908,A -85,B 0,C 180,E1 -3306.808,E2 -3306.808} C_VEL
LIN {X 0,Y 552.876,Z 229.71,A -85,B 0,C 180,E1 -3309.928,E2 -3309.928} C_VEL
LIN {X 0,Y 552.615,Z 251.419,A -85,B 0,C 180,E1 -3312.992,E2 -3312.992} C_VEL
LIN {X 0,Y 552.377,Z 270.276,A -85,B 0,C 180,E1 -3315.625,E2 -3315.625} C_VEL
LIN {X 0,Y 553.423,Z 278.492,A -85,B 0,C 180,E1 -3315.762,E2 -3315.762} C_VEL
LIN {X 0,Y 553.128,Z 378.853,A -85,B 0,C 180,E1 -3317.083,E2 -3317.083} C_VEL
LIN {X 0,Y 552.981,Z 392.158,A -85,B 0,C 180,E1 -3317.406,E2 -3317.406} C_VEL
LIN {X 0,Y 552.853,Z 405.146,A -85,B 0,C 180,E1 -3317.878,E2 -3317.878} C_VEL
LIN {X 0,Y 552.684,Z 417.621,A -85,B 0,C 180,E1 -3318.506,E2 -3318.506} C_VEL
LIN {X 0,Y 552.471,Z 429.48,A -85,B 0,C 180,E1 -3319.278,E2 -3319.278} C_VEL
LIN {X 0,Y 552.284,Z 439.642,A -85,B 0,C 180,E1 -3320.108,E2 -3320.108} C_VEL
LIN {X 0,Y 552.104,Z 448.782,A -85,B 0,C 180,E1 -3321.028,E2 -3321.028} C_VEL
LIN {X 0,Y 551.961,Z 457.684,A -85,B 0,C 180,E1 -3322.132,E2 -3322.132} C_VEL
LIN {X 0,Y 551.836,Z 464.845,A -85,B 0,C 180,E1 -3323.234,E2 -3323.234} C_VEL
LIN {X 0,Y 551.804,Z 471.363,A -85,B 0,C 180,E1 -3324.518,E2 -3324.518} C_VEL
LIN {X 0,Y 551.764,Z 475.674,A -85,B 0,C 180,E1 -3325.616,E2 -3325.616} C_VEL
LIN {X 0,Y 551.751,Z 477.955,A -85,B 0,C 180,E1 -3326.348,E2 -3326.348} C_VEL
LIN {X 0,Y 551.724,Z 479.805,A -85,B 0,C 180,E1 -3327.078,E2 -3327.078} C_VEL
LIN {X 0,Y 551.645,Z 482.181,A -85,B 0,C 180,E1 -3328.539,E2 -3328.539} C_VEL
LIN {X 0,Y 551.64,Z 483,A -85,B 0,C 180,E1 -3329.999,E2 -3329.999} C_VEL
LIN {X 0,Y 551.645,Z 482.185,A -85,B 0,C 180,E1 -3331.459,E2 -3331.459} C_VEL
LIN {X 0,Y 551.723,Z 479.813,A -85,B 0,C 180,E1 -3332.919,E2 -3332.919} C_VEL
LIN {X 0,Y 551.763,Z 476.9,A -85,B 0,C 180,E1 -3334.016,E2 -3334.016} C_VEL
LIN {X 0,Y 551.723,Z 472.955,A -85,B 0,C 180,E1 -3335.114,E2 -3335.114} C_VEL
LIN {X 0,Y 551.814,Z 467.13,A -85,B 0,C 180,E1 -3336.352,E2 -3336.352} C_VEL
LIN {X 0,Y 551.925,Z 460.249,A -85,B 0,C 180,E1 -3337.498,E2 -3337.498} C_VEL
LIN {X 0,Y 552.081,Z 452.009,A -85,B 0,C 180,E1 -3338.6,E2 -3338.6} C_VEL
LIN {X 0,Y 552.223,Z 443.562,A -85,B 0,C 180,E1 -3339.521,E2 -3339.521} C_VEL
LIN {X 0,Y 552.426,Z 433.119,A -85,B 0,C 180,E1 -3340.443,E2 -3340.443} C_VEL
LIN {X 0,Y 552.59,Z 422.162,A -85,B 0,C 180,E1 -3341.222,E2 -3341.222} C_VEL
LIN {X 0,Y 552.747,Z 411.449,A -85,B 0,C 180,E1 -3341.829,E2 -3341.829} C_VEL
LIN {X 0,Y 552.886,Z 399.803,A -85,B 0,C 180,E1 -3342.338,E2 -3342.338} C_VEL
LIN {X 0,Y 553.059,Z 387.29,A -85,B 0,C 180,E1 -3342.73,E2 -3342.73} C_VEL
LIN {X 0,Y 553.137,Z 374.664,A -85,B 0,C 180,E1 -3342.985,E2 -3342.985} C_VEL
LIN {X 0,Y 553.255,Z 276.242,A -85,B 0,C 180,E1 -3344.272,E2 -3344.272} C_VEL
LIN {X 0,Y 552.39,Z 270.229,A -85,B 0,C 180,E1 -3344.386,E2 -3344.386} C_VEL
LIN {X 0,Y 552.63,Z 248.115,A -85,B 0,C 180,E1 -3347.483,E2 -3347.483} C_VEL
LIN {X 0,Y 552.935,Z 227.136,A -85,B 0,C 180,E1 -3350.456,E2 -3350.456} C_VEL
LIN {X 0,Y 553.225,Z 208.172,A -85,B 0,C 180,E1 -3353.188,E2 -3353.188} C_VEL
LIN {X 0,Y 552.166,Z 200.75,A -85,B 0,C 180,E1 -3354.319,E2 -3354.319} C_VEL
LIN {X 0,Y 552.131,Z 200.706,A -85,B 0,C 180,E1 -3357.269,E2 -3357.269} C_VEL
LIN {X 0,Y 552.103,Z 200.717,A -85,B 0,C 180,E1 -3360.048,E2 -3360.048} C_VEL
LIN {X 0,Y 552.111,Z 200.707,A -85,B 0,C 180,E1 -3362.845,E2 -3362.845} C_VEL
LIN {X 0,Y 552.085,Z 200.711,A -85,B 0,C 180,E1 -3365.44,E2 -3365.44} C_VEL
LIN {X 0,Y 552.074,Z 200.719,A -85,B 0,C 180,E1 -3367.882,E2 -3367.882} C_VEL
LIN {X 0,Y 552.096,Z 200.71,A -85,B 0,C 180,E1 -3370.476,E2 -3370.476} C_VEL
LIN {X 0,Y 552.075,Z 200.714,A -85,B 0,C 180,E1 -3373.479,E2 -3373.479} C_VEL
LIN {X 0,Y 552.091,Z 200.709,A -85,B 0,C 180,E1 -3376.574,E2 -3376.574} C_VEL
LIN {X 0,Y 552.121,Z 200.711,A -85,B 0,C 180,E1 -3379.52,E2 -3379.52} C_VEL
LIN {X 0,Y 552.056,Z 200.714,A -85,B 0,C 180,E1 -3382.333,E2 -3382.333} C_VEL
LIN {X 0,Y 552.091,Z 200.71,A -85,B 0,C 180,E1 -3385.051,E2 -3385.051} C_VEL
LIN {X 0,Y 552.088,Z 200.718,A -85,B 0,C 180,E1 -3387.679,E2 -3387.679} C_VEL
LIN {X 0,Y 552.105,Z 200.708,A -85,B 0,C 180,E1 -3390.234,E2 -3390.234} C_VEL
LIN {X 0,Y 552.1,Z 200.71,A -85,B 0,C 180,E1 -3392.995,E2 -3392.995} C_VEL
LIN {X 0,Y 552.069,Z 200.716,A -85,B 0,C 180,E1 -3395.159,E2 -3395.159} C_VEL
LIN {X 0,Y 552.077,Z 200.719,A -85,B 0,C 180,E1 -3397.548,E2 -3397.548} C_VEL
LIN {X 0,Y 552.106,Z 200.707,A -85,B 0,C 180,E1 -3400.672,E2 -3400.672} C_VEL
LIN {X 0,Y 552.14,Z 200.706,A -85,B 0,C 180,E1 -3402.977,E2 -3402.977} C_VEL
LIN {X 0,Y 552.091,Z 200.71,A -85,B 0,C 180,E1 -3406.003,E2 -3406.003} C_VEL
LIN {X 0,Y 552.157,Z 200.706,A -85,B 0,C 180,E1 -3408.993,E2 -3408.993} C_VEL
LIN {X 0,Y 552.11,Z 200.707,A -85,B 0,C 180,E1 -3411.951,E2 -3411.951} C_VEL
LIN {X 0,Y 552.152,Z 200.701,A -85,B 0,C 180,E1 -3414.155,E2 -3414.155} C_VEL
LIN {X 0,Y 552.161,Z 200.709,A -85,B 0,C 180,E1 -3417.081,E2 -3417.081} C_VEL
LIN {X 0,Y 552.167,Z 200.699,A -85,B 0,C 180,E1 -3420,E2 -3420} C_VEL
LIN {X 0,Y 552.158,Z 200.708,A -85,B 0,C 180,E1 -3422.918,E2 -3422.918} C_VEL
LIN {X 0,Y 552.142,Z 200.702,A -85,B 0,C 180,E1 -3425.844,E2 -3425.844} C_VEL
LIN {X 0,Y 552.114,Z 200.713,A -85,B 0,C 180,E1 -3428.786,E2 -3428.786} C_VEL
LIN {X 0,Y 552.109,Z 200.706,A -85,B 0,C 180,E1 -3431.751,E2 -3431.751} C_VEL
LIN {X 0,Y 552.08,Z 200.719,A -85,B 0,C 180,E1 -3434.75,E2 -3434.75} C_VEL
LIN {X 0,Y 552.087,Z 200.709,A -85,B 0,C 180,E1 -3437.789,E2 -3437.789} C_VEL
LIN {X 0,Y 552.082,Z 200.711,A -85,B 0,C 180,E1 -3440.103,E2 -3440.103} C_VEL
LIN {X 0,Y 552.061,Z 200.718,A -85,B 0,C 180,E1 -3442.452,E2 -3442.452} C_VEL
LIN {X 0,Y 552.105,Z 200.708,A -85,B 0,C 180,E1 -3445.353,E2 -3445.353} C_VEL
LIN {X 0,Y 552.084,Z 200.712,A -85,B 0,C 180,E1 -3448.099,E2 -3448.099} C_VEL
LIN {X 0,Y 552.058,Z 200.721,A -85,B 0,C 180,E1 -3450.644,E2 -3450.644} C_VEL
LIN {X 0,Y 552.076,Z 200.711,A -85,B 0,C 180,E1 -3453.188,E2 -3453.188} C_VEL
LIN {X 0,Y 552.07,Z 200.712,A -85,B 0,C 180,E1 -3453.824,E2 -3453.824} C_VEL
LIN {X 0,Y 551.438,Z 200.799,A -85,B 0,C 180,E1 -3454.433,E2 -3454.433} C_VEL
LIN {X 0,Y 548.618,Z 201.149,A -85,B 0,C 180,E1 -3455.421,E2 -3455.421} C_VEL
LIN {X 0,Y 546.197,Z 201.45,A -85,B 0,C 180,E1 -3456.216,E2 -3456.216} C_VEL
LIN {X 0,Y 545.126,Z 201.581,A -85,B 0,C 180,E1 -3456.83,E2 -3456.83} C_VEL
LIN {X 0,Y 545.023,Z 201.591,A -85,B 0,C 180,E1 -3457.038,E2 -3457.038} C_VEL
LIN {X 0,Y 545.032,Z 201.594,A -85,B 0,C 180,E1 -3460.145,E2 -3460.145} C_VEL
LIN {X 0,Y 545.027,Z 201.593,A -85,B 0,C 180,E1 -3462.7,E2 -3462.7} C_VEL
LIN {X 0,Y 545.001,Z 201.592,A -85,B 0,C 180,E1 -3465.173,E2 -3465.173} C_VEL
LIN {X 0,Y 545.051,Z 201.59,A -85,B 0,C 180,E1 -3467.901,E2 -3467.901} C_VEL
LIN {X 0,Y 545.053,Z 201.587,A -85,B 0,C 180,E1 -3470.822,E2 -3470.822} C_VEL
LIN {X 0,Y 545.027,Z 201.591,A -85,B 0,C 180,E1 -3473.624,E2 -3473.624} C_VEL
LIN {X 0,Y 545.043,Z 201.593,A -85,B 0,C 180,E1 -3476.332,E2 -3476.332} C_VEL
LIN {X 0,Y 545.046,Z 201.586,A -85,B 0,C 180,E1 -3478.956,E2 -3478.956} C_VEL
LIN {X 0,Y 545.082,Z 201.584,A -85,B 0,C 180,E1 -3481.511,E2 -3481.511} C_VEL
LIN {X 0,Y 545.08,Z 201.584,A -85,B 0,C 180,E1 -3484.494,E2 -3484.494} C_VEL
LIN {X 0,Y 545.023,Z 201.59,A -85,B 0,C 180,E1 -3487.245,E2 -3487.245} C_VEL
LIN {X 0,Y 545.105,Z 201.581,A -85,B 0,C 180,E1 -3490.418,E2 -3490.418} C_VEL
LIN {X 0,Y 545.038,Z 201.592,A -85,B 0,C 180,E1 -3493.523,E2 -3493.523} C_VEL
LIN {X 0,Y 545.075,Z 201.592,A -85,B 0,C 180,E1 -3495.822,E2 -3495.822} C_VEL
LIN {X 0,Y 545.112,Z 201.578,A -85,B 0,C 180,E1 -3498.852,E2 -3498.852} C_VEL
LIN {X 0,Y 545.12,Z 201.585,A -85,B 0,C 180,E1 -3501.849,E2 -3501.849} C_VEL
LIN {X 0,Y 545.194,Z 201.571,A -85,B 0,C 180,E1 -3504.825,E2 -3504.825} C_VEL
LIN {X 0,Y 545.052,Z 201.598,A -85,B 0,C 180,E1 -3506.398,E2 -3506.398} C_VEL
LIN {X 0,Y 545.363,Z 206.914,A -85,B 0,C 180,E1 -3507.416,E2 -3507.416} C_VEL
LIN {X 0,Y 545.242,Z 220.535,A -85,B 0,C 180,E1 -3510.001,E2 -3510.001} C_VEL
LIN {X 0,Y 545.167,Z 223.094,A -85,B 0,C 180,E1 -3510.486,E2 -3510.486} C_VEL
LIN {X 0,Y 546.575,Z 230.939,A -85,B 0,C 180,E1 -3510.646,E2 -3510.646} C_VEL
LIN {X 0,Y 546.211,Z 329.355,A -85,B 0,C 180,E1 -3511.96,E2 -3511.96} C_VEL
LIN {X 0,Y 546.075,Z 341.765,A -85,B 0,C 180,E1 -3512.26,E2 -3512.26} C_VEL
LIN {X 0,Y 545.921,Z 354.548,A -85,B 0,C 180,E1 -3512.722,E2 -3512.722} C_VEL
LIN {X 0,Y 545.716,Z 366.751,A -85,B 0,C 180,E1 -3513.323,E2 -3513.323} C_VEL
LIN {X 0,Y 545.481,Z 378.245,A -85,B 0,C 180,E1 -3514.064,E2 -3514.064} C_VEL
LIN {X 0,Y 545.297,Z 388.588,A -85,B 0,C 180,E1 -3514.899,E2 -3514.899} C_VEL
LIN {X 0,Y 545.07,Z 397.093,A -85,B 0,C 180,E1 -3515.736,E2 -3515.736} C_VEL
LIN {X 0,Y 544.959,Z 405.751,A -85,B 0,C 180,E1 -3516.775,E2 -3516.775} C_VEL
LIN {X 0,Y 544.83,Z 413.72,A -85,B 0,C 180,E1 -3517.971,E2 -3517.971} C_VEL
LIN {X 0,Y 544.713,Z 420.584,A -85,B 0,C 180,E1 -3519.281,E2 -3519.281} C_VEL
LIN {X 0,Y 544.653,Z 425.115,A -85,B 0,C 180,E1 -3520.408,E2 -3520.408} C_VEL
LIN {X 0,Y 544.634,Z 427.823,A -85,B 0,C 180,E1 -3521.273,E2 -3521.273} C_VEL
LIN {X 0,Y 544.569,Z 431.001,A -85,B 0,C 180,E1 -3522.674,E2 -3522.674} C_VEL
LIN {X 0,Y 544.555,Z 432.071,A -85,B 0,C 180,E1 -3523.433,E2 -3523.433} C_VEL
LIN {X 0,Y 544.589,Z 432.924,A -85,B 0,C 180,E1 -3524.561,E2 -3524.561} C_VEL
LIN {X 0,Y 544.528,Z 432.849,A -85,B 0,C 180,E1 -3525.726,E2 -3525.726} C_VEL
LIN {X 0,Y 544.554,Z 432.243,A -85,B 0,C 180,E1 -3526.495,E2 -3526.495} C_VEL
LIN {X 0,Y 544.575,Z 431.228,A -85,B 0,C 180,E1 -3527.267,E2 -3527.267} C_VEL
LIN {X 0,Y 544.574,Z 429.775,A -85,B 0,C 180,E1 -3528.043,E2 -3528.043} C_VEL
LIN {X 0,Y 544.635,Z 426.679,A -85,B 0,C 180,E1 -3529.211,E2 -3529.211} C_VEL
LIN {X 0,Y 544.684,Z 422.405,A -85,B 0,C 180,E1 -3530.388,E2 -3530.388} C_VEL
LIN {X 0,Y 544.762,Z 415.897,A -85,B 0,C 180,E1 -3531.741,E2 -3531.741} C_VEL
LIN {X 0,Y 544.88,Z 409.661,A -85,B 0,C 180,E1 -3532.764,E2 -3532.764} C_VEL
LIN {X 0,Y 545.02,Z 401.972,A -85,B 0,C 180,E1 -3533.798,E2 -3533.798} C_VEL
LIN {X 0,Y 545.195,Z 392.054,A -85,B 0,C 180,E1 -3534.869,E2 -3534.869} C_VEL
LIN {X 0,Y 545.383,Z 382.222,A -85,B 0,C 180,E1 -3535.728,E2 -3535.728} C_VEL
LIN {X 0,Y 545.618,Z 371.48,A -85,B 0,C 180,E1 -3536.486,E2 -3536.486} C_VEL
LIN {X 0,Y 545.835,Z 360.406,A -85,B 0,C 180,E1 -3537.101,E2 -3537.101} C_VEL
LIN {X 0,Y 545.984,Z 347.151,A -85,B 0,C 180,E1 -3537.657,E2 -3537.657} C_VEL
LIN {X 0,Y 546.114,Z 334.959,A -85,B 0,C 180,E1 -3538.015,E2 -3538.015} C_VEL
LIN {X 0,Y 546.188,Z 321.925,A -85,B 0,C 180,E1 -3538.246,E2 -3538.246} C_VEL
LIN {X 0,Y 546.462,Z 230.403,A -85,B 0,C 180,E1 -3539.454,E2 -3539.454} C_VEL
LIN {X 0,Y 545.169,Z 223.032,A -85,B 0,C 180,E1 -3539.606,E2 -3539.606} C_VEL
LIN {X 0,Y 545.304,Z 213.681,A -85,B 0,C 180,E1 -3541.374,E2 -3541.374} C_VEL
LIN {X 0,Y 545.21,Z 201.806,A -85,B 0,C 180,E1 -3543.575,E2 -3543.575} C_VEL
LIN {X 0,Y 545.147,Z 201.58,A -85,B 0,C 180,E1 -3543.664,E2 -3543.664} C_VEL
LIN {X 0,Y 545.068,Z 201.588,A -85,B 0,C 180,E1 -3546.926,E2 -3546.926} C_VEL
LIN {X 0,Y 545.08,Z 201.59,A -85,B 0,C 180,E1 -3550.139,E2 -3550.139} C_VEL
LIN {X 0,Y 545.053,Z 201.591,A -85,B 0,C 180,E1 -3552.696,E2 -3552.696} C_VEL
LIN {X 0,Y 545.046,Z 201.588,A -85,B 0,C 180,E1 -3555.165,E2 -3555.165} C_VEL
LIN {X 0,Y 545.065,Z 201.59,A -85,B 0,C 180,E1 -3557.896,E2 -3557.896} C_VEL
LIN {X 0,Y 545.086,Z 201.584,A -85,B 0,C 180,E1 -3560.674,E2 -3560.674} C_VEL
LIN {X 0,Y 545.033,Z 201.591,A -85,B 0,C 180,E1 -3563.619,E2 -3563.619} C_VEL
LIN {X 0,Y 545.054,Z 201.59,A -85,B 0,C 180,E1 -3566.328,E2 -3566.328} C_VEL
LIN {X 0,Y 545.045,Z 201.586,A -85,B 0,C 180,E1 -3568.951,E2 -3568.951} C_VEL
LIN {X 0,Y 545.085,Z 201.585,A -85,B 0,C 180,E1 -3571.507,E2 -3571.507} C_VEL
LIN {X 0,Y 545.07,Z 201.583,A -85,B 0,C 180,E1 -3574.489,E2 -3574.489} C_VEL
LIN {X 0,Y 545.046,Z 201.588,A -85,B 0,C 180,E1 -3577.243,E2 -3577.243} C_VEL
LIN {X 0,Y 545.089,Z 201.582,A -85,B 0,C 180,E1 -3580.414,E2 -3580.414} C_VEL
LIN {X 0,Y 545.117,Z 201.576,A -85,B 0,C 180,E1 -3582.751,E2 -3582.751} C_VEL
LIN {X 0,Y 545.065,Z 201.589,A -85,B 0,C 180,E1 -3585.819,E2 -3585.819} C_VEL
LIN {X 0,Y 545.1,Z 201.58,A -85,B 0,C 180,E1 -3588.849,E2 -3588.849} C_VEL
LIN {X 0,Y 545.102,Z 201.581,A -85,B 0,C 180,E1 -3591.847,E2 -3591.847} C_VEL
LIN {X 0,Y 545.142,Z 201.575,A -85,B 0,C 180,E1 -3594.08,E2 -3594.08} C_VEL
LIN {X 0,Y 545.146,Z 201.577,A -85,B 0,C 180,E1 -3597.044,E2 -3597.044} C_VEL
LIN {X 0,Y 545.158,Z 201.571,A -85,B 0,C 180,E1 -3600,E2 -3600} C_VEL
LIN {X 0,Y 545.142,Z 201.578,A -85,B 0,C 180,E1 -3602.956,E2 -3602.956} C_VEL
LIN {X 0,Y 545.133,Z 201.573,A -85,B 0,C 180,E1 -3605.92,E2 -3605.92} C_VEL
LIN {X 0,Y 545.075,Z 201.589,A -85,B 0,C 180,E1 -3608.901,E2 -3608.901} C_VEL
LIN {X 0,Y 545.102,Z 201.579,A -85,B 0,C 180,E1 -3611.905,E2 -3611.905} C_VEL
LIN {X 0,Y 545.051,Z 201.592,A -85,B 0,C 180,E1 -3614.945,E2 -3614.945} C_VEL
LIN {X 0,Y 545.036,Z 201.587,A -85,B 0,C 180,E1 -3618.027,E2 -3618.027} C_VEL
LIN {X 0,Y 545.063,Z 201.586,A -85,B 0,C 180,E1 -3620.374,E2 -3620.374} C_VEL
LIN {X 0,Y 545.041,Z 201.586,A -85,B 0,C 180,E1 -3623.561,E2 -3623.561} C_VEL
LIN {X 0,Y 545.056,Z 201.591,A -85,B 0,C 180,E1 -3626.827,E2 -3626.827} C_VEL
LIN {X 0,Y 545.028,Z 201.59,A -85,B 0,C 180,E1 -3629.341,E2 -3629.341} C_VEL
LIN {X 0,Y 545.029,Z 201.589,A -85,B 0,C 180,E1 -3631.917,E2 -3631.917} C_VEL
LIN {X 0,Y 545.034,Z 201.596,A -85,B 0,C 180,E1 -3634.567,E2 -3634.567} C_VEL
LIN {X 0,Y 545.008,Z 201.591,A -85,B 0,C 180,E1 -3637.307,E2 -3637.307} C_VEL
LIN {X 0,Y 545.045,Z 201.593,A -85,B 0,C 180,E1 -3640.145,E2 -3640.145} C_VEL
LIN {X 0,Y 545.063,Z 201.585,A -85,B 0,C 180,E1 -3643.109,E2 -3643.109} C_VEL
LIN {X 0,Y 545.035,Z 201.597,A -85,B 0,C 180,E1 -3646.228,E2 -3646.228} C_VEL
LIN {X 0,Y 545.059,Z 201.586,A -85,B 0,C 180,E1 -3648.886,E2 -3648.886} C_VEL
LIN {X 0,Y 545.037,Z 201.594,A -85,B 0,C 180,E1 -3651.866,E2 -3651.866} C_VEL
LIN {X 0,Y 545.042,Z 201.591,A -85,B 0,C 180,E1 -3654.534,E2 -3654.534} C_VEL
LIN {X 0,Y 545.062,Z 201.586,A -85,B 0,C 180,E1 -3657.213,E2 -3657.213} C_VEL
LIN {X 0,Y 545.057,Z 201.593,A -85,B 0,C 180,E1 -3659.812,E2 -3659.812} C_VEL
LIN {X 0,Y 545.048,Z 201.592,A -85,B 0,C 180,E1 -3662.343,E2 -3662.343} C_VEL
LIN {X 0,Y 545.092,Z 201.589,A -85,B 0,C 180,E1 -3665.431,E2 -3665.431} C_VEL
LIN {X 0,Y 545.105,Z 201.67,A -85,B 0,C 180,E1 -3665.584,E2 -3665.584} C_VEL
LIN {X 0,Y 546.236,Z 208.909,A -85,B 0,C 180,E1 -3666.695,E2 -3666.695} C_VEL
LIN {X 0,Y 545.952,Z 229.355,A -85,B 0,C 180,E1 -3669.662,E2 -3669.662} C_VEL
LIN {X 0,Y 545.598,Z 251.069,A -85,B 0,C 180,E1 -3672.767,E2 -3672.767} C_VEL
LIN {X 0,Y 545.324,Z 269.922,A -85,B 0,C 180,E1 -3675.433,E2 -3675.433} C_VEL
LIN {X 0,Y 546.531,Z 278.978,A -85,B 0,C 180,E1 -3675.59,E2 -3675.59} C_VEL
LIN {X 0,Y 546.205,Z 378.473,A -85,B 0,C 180,E1 -3676.916,E2 -3676.916} C_VEL
LIN {X 0,Y 546.019,Z 391.791,A -85,B 0,C 180,E1 -3677.242,E2 -3677.242} C_VEL
LIN {X 0,Y 545.897,Z 403.994,A -85,B 0,C 180,E1 -3677.688,E2 -3677.688} C_VEL
LIN {X 0,Y 545.702,Z 416.197,A -85,B 0,C 180,E1 -3678.29,E2 -3678.29} C_VEL
LIN {X 0,Y 545.496,Z 427.943,A -85,B 0,C 180,E1 -3679.045,E2 -3679.045} C_VEL
LIN {X 0,Y 545.265,Z 438.419,A -85,B 0,C 180,E1 -3679.885,E2 -3679.885} C_VEL
LIN {X 0,Y 545.086,Z 446.987,A -85,B 0,C 180,E1 -3680.725,E2 -3680.725} C_VEL
LIN {X 0,Y 544.978,Z 454.897,A -85,B 0,C 180,E1 -3681.658,E2 -3681.658} C_VEL
LIN {X 0,Y 544.824,Z 462.613,A -85,B 0,C 180,E1 -3682.774,E2 -3682.774} C_VEL
LIN {X 0,Y 544.777,Z 469.676,A -85,B 0,C 180,E1 -3684.075,E2 -3684.075} C_VEL
LIN {X 0,Y 544.629,Z 474.37,A -85,B 0,C 180,E1 -3685.188,E2 -3685.188} C_VEL
LIN {X 0,Y 544.669,Z 477.955,A -85,B 0,C 180,E1 -3686.3,E2 -3686.3} C_VEL
LIN {X 0,Y 544.651,Z 479.804,A -85,B 0,C 180,E1 -3687.04,E2 -3687.04} C_VEL
LIN {X 0,Y 544.546,Z 482.18,A -85,B 0,C 180,E1 -3688.52,E2 -3688.52} C_VEL
LIN {X 0,Y 544.541,Z 483,A -85,B 0,C 180,E1 -3689.999,E2 -3689.999} C_VEL
LIN {X 0,Y 544.546,Z 482.185,A -85,B 0,C 180,E1 -3691.478,E2 -3691.478} C_VEL
LIN {X 0,Y 544.65,Z 479.813,A -85,B 0,C 180,E1 -3692.957,E2 -3692.957} C_VEL
LIN {X 0,Y 544.683,Z 476.9,A -85,B 0,C 180,E1 -3694.068,E2 -3694.068} C_VEL
LIN {X 0,Y 544.653,Z 472.955,A -85,B 0,C 180,E1 -3695.181,E2 -3695.181} C_VEL
LIN {X 0,Y 544.729,Z 467.649,A -85,B 0,C 180,E1 -3696.339,E2 -3696.339} C_VEL
LIN {X 0,Y 544.834,Z 461.469,A -85,B 0,C 180,E1 -3697.409,E2 -3697.409} C_VEL
LIN {X 0,Y 545.005,Z 453.425,A -85,B 0,C 180,E1 -3698.526,E2 -3698.526} C_VEL
LIN {X 0,Y 545.124,Z 445.223,A -85,B 0,C 180,E1 -3699.459,E2 -3699.459} C_VEL
LIN {X 0,Y 545.374,Z 435.23,A -85,B 0,C 180,E1 -3700.391,E2 -3700.391} C_VEL
LIN {X 0,Y 545.56,Z 424.315,A -85,B 0,C 180,E1 -3701.209,E2 -3701.209} C_VEL
LIN {X 0,Y 545.737,Z 412.901,A -85,B 0,C 180,E1 -3701.888,E2 -3701.888} C_VEL
LIN {X 0,Y 545.919,Z 400.663,A -85,B 0,C 180,E1 -3702.45,E2 -3702.45} C_VEL
LIN {X 0,Y 546.112,Z 387.851,A -85,B 0,C 180,E1 -3702.871,E2 -3702.871} C_VEL
LIN {X 0,Y 546.232,Z 374.29,A -85,B 0,C 180,E1 -3703.152,E2 -3703.152} C_VEL
LIN {X 0,Y 546.414,Z 277.318,A -85,B 0,C 180,E1 -3704.436,E2 -3704.436} C_VEL
LIN {X 0,Y 545.368,Z 269.947,A -85,B 0,C 180,E1 -3704.569,E2 -3704.569} C_VEL
LIN {X 0,Y 545.621,Z 248.591,A -85,B 0,C 180,E1 -3707.602,E2 -3707.602} C_VEL
LIN {X 0,Y 545.993,Z 226.826,A -85,B 0,C 180,E1 -3710.728,E2 -3710.728} C_VEL
LIN {X 0,Y 546.273,Z 209.232,A -85,B 0,C 180,E1 -3713.3,E2 -3713.3} C_VEL
LIN {X 0,Y 545.118,Z 201.632,A -85,B 0,C 180,E1 -3714.476,E2 -3714.476} C_VEL
LIN {X 0,Y 545.078,Z 201.587,A -85,B 0,C 180,E1 -3717.652,E2 -3717.652} C_VEL
LIN {X 0,Y 545.061,Z 201.592,A -85,B 0,C 180,E1 -3720.243,E2 -3720.243} C_VEL
LIN {X 0,Y 545.073,Z 201.583,A -85,B 0,C 180,E1 -3723.061,E2 -3723.061} C_VEL
LIN {X 0,Y 545.041,Z 201.591,A -85,B 0,C 180,E1 -3725.673,E2 -3725.673} C_VEL
LIN {X 0,Y 545.03,Z 201.593,A -85,B 0,C 180,E1 -3728.233,E2 -3728.233} C_VEL
LIN {X 0,Y 545.07,Z 201.584,A -85,B 0,C 180,E1 -3731.109,E2 -3731.109} C_VEL
LIN {X 0,Y 545.025,Z 201.594,A -85,B 0,C 180,E1 -3734.126,E2 -3734.126} C_VEL
LIN {X 0,Y 545.056,Z 201.585,A -85,B 0,C 180,E1 -3736.891,E2 -3736.891} C_VEL
LIN {X 0,Y 545.088,Z 201.587,A -85,B 0,C 180,E1 -3739.518,E2 -3739.518} C_VEL
LIN {X 0,Y 545.016,Z 201.597,A -85,B 0,C 180,E1 -3741.86,E2 -3741.86} C_VEL
LIN {X 0,Y 545.025,Z 201.589,A -85,B 0,C 180,E1 -3744.53,E2 -3744.53} C_VEL
LIN {X 0,Y 545.042,Z 201.59,A -85,B 0,C 180,E1 -3747.209,E2 -3747.209} C_VEL
LIN {X 0,Y 545.057,Z 201.591,A -85,B 0,C 180,E1 -3749.81,E2 -3749.81} C_VEL
LIN {X 0,Y 545.055,Z 201.585,A -85,B 0,C 180,E1 -3752.342,E2 -3752.342} C_VEL
LIN {X 0,Y 545.07,Z 201.584,A -85,B 0,C 180,E1 -3754.818,E2 -3754.818} C_VEL
LIN {X 0,Y 545.03,Z 201.594,A -85,B 0,C 180,E1 -3757.242,E2 -3757.242} C_VEL
LIN {X 0,Y 545.068,Z 201.583,A -85,B 0,C 180,E1 -3760.413,E2 -3760.413} C_VEL
LIN {X 0,Y 545.095,Z 201.581,A -85,B 0,C 180,E1 -3762.75,E2 -3762.75} C_VEL
LIN {X 0,Y 545.046,Z 201.589,A -85,B 0,C 180,E1 -3765.818,E2 -3765.818} C_VEL
LIN {X 0,Y 545.103,Z 201.583,A -85,B 0,C 180,E1 -3768.849,E2 -3768.849} C_VEL
LIN {X 0,Y 545.08,Z 201.583,A -85,B 0,C 180,E1 -3771.846,E2 -3771.846} C_VEL
LIN {X 0,Y 545.125,Z 201.576,A -85,B 0,C 180,E1 -3774.08,E2 -3774.08} C_VEL
LIN {X 0,Y 545.127,Z 201.585,A -85,B 0,C 180,E1 -3777.044,E2 -3777.044} C_VEL
LIN {X 0,Y 545.137,Z 201.575,A -85,B 0,C 180,E1 -3780,E2 -3780} C_VEL
LIN {X 0,Y 545.124,Z 201.585,A -85,B 0,C 180,E1 -3782.956,E2 -3782.956} C_VEL
LIN {X 0,Y 545.113,Z 201.578,A -85,B 0,C 180,E1 -3785.92,E2 -3785.92} C_VEL
LIN {X 0,Y 545.071,Z 201.593,A -85,B 0,C 180,E1 -3788.901,E2 -3788.901} C_VEL
LIN {X 0,Y 545.079,Z 201.582,A -85,B 0,C 180,E1 -3791.905,E2 -3791.905} C_VEL
LIN {X 0,Y 545.029,Z 201.596,A -85,B 0,C 180,E1 -3794.945,E2 -3794.945} C_VEL
LIN {X 0,Y 545.087,Z 201.582,A -85,B 0,C 180,E1 -3797.447,E2 -3797.447} C_VEL
LIN {X 0,Y 545.047,Z 201.59,A -85,B 0,C 180,E1 -3800.374,E2 -3800.374} C_VEL
LIN {X 0,Y 545.061,Z 201.584,A -85,B 0,C 180,E1 -3803.56,E2 -3803.56} C_VEL
LIN {X 0,Y 545.037,Z 201.589,A -85,B 0,C 180,E1 -3806.003,E2 -3806.003} C_VEL
LIN {X 0,Y 545.048,Z 201.593,A -85,B 0,C 180,E1 -3808.752,E2 -3808.752} C_VEL
LIN {X 0,Y 545.026,Z 201.59,A -85,B 0,C 180,E1 -3811.916,E2 -3811.916} C_VEL
LIN {X 0,Y 545.037,Z 201.596,A -85,B 0,C 180,E1 -3814.566,E2 -3814.566} C_VEL
LIN {X 0,Y 545.023,Z 201.591,A -85,B 0,C 180,E1 -3817.038,E2 -3817.038} C_VEL
LIN {X 0,Y 544.314,Z 201.678,A -85,B 0,C 180,E1 -3817.655,E2 -3817.655} C_VEL
LIN {X 0,Y 541.448,Z 202.04,A -85,B 0,C 180,E1 -3818.656,E2 -3818.656} C_VEL
LIN {X 0,Y 539.063,Z 202.334,A -85,B 0,C 180,E1 -3819.461,E2 -3819.461} C_VEL
LIN {X 0,Y 538.057,Z 202.462,A -85,B 0,C 180,E1 -3820.083,E2 -3820.083} C_VEL
LIN {X 0,Y 537.984,Z 202.466,A -85,B 0,C 180,E1 -3820.294,E2 -3820.294} C_VEL
LIN {X 0,Y 537.99,Z 202.466,A -85,B 0,C 180,E1 -3822.991,E2 -3822.991} C_VEL
LIN {X 0,Y 537.976,Z 202.475,A -85,B 0,C 180,E1 -3826.188,E2 -3826.188} C_VEL
LIN {X 0,Y 538.022,Z 202.461,A -85,B 0,C 180,E1 -3829.256,E2 -3829.256} C_VEL
LIN {X 0,Y 537.965,Z 202.477,A -85,B 0,C 180,E1 -3832.126,E2 -3832.126} C_VEL
LIN {X 0,Y 537.989,Z 202.466,A -85,B 0,C 180,E1 -3834.92,E2 -3834.92} C_VEL
LIN {X 0,Y 537.997,Z 202.467,A -85,B 0,C 180,E1 -3837.621,E2 -3837.621} C_VEL
LIN {X 0,Y 537.998,Z 202.471,A -85,B 0,C 180,E1 -3840.242,E2 -3840.242} C_VEL
LIN {X 0,Y 538.036,Z 202.46,A -85,B 0,C 180,E1 -3842.799,E2 -3842.799} C_VEL
LIN {X 0,Y 538.013,Z 202.463,A -85,B 0,C 180,E1 -3845.295,E2 -3845.295} C_VEL
LIN {X 0,Y 538.003,Z 202.471,A -85,B 0,C 180,E1 -3848.045,E2 -3848.045} C_VEL
LIN {X 0,Y 538.069,Z 202.461,A -85,B 0,C 180,E1 -3850.151,E2 -3850.151} C_VEL
LIN {X 0,Y 537.987,Z 202.468,A -85,B 0,C 180,E1 -3853.301,E2 -3853.301} C_VEL
LIN {X 0,Y 538.044,Z 202.466,A -85,B 0,C 180,E1 -3855.633,E2 -3855.633} C_VEL
LIN {X 0,Y 538.071,Z 202.455,A -85,B 0,C 180,E1 -3858.704,E2 -3858.704} C_VEL
LIN {X 0,Y 538.077,Z 202.464,A -85,B 0,C 180,E1 -3861.742,E2 -3861.742} C_VEL
LIN {X 0,Y 538.152,Z 202.448,A -85,B 0,C 180,E1 -3864.757,E2 -3864.757} C_VEL
LIN {X 0,Y 538.001,Z 202.564,A -85,B 0,C 180,E1 -3866.327,E2 -3866.327} C_VEL
LIN {X 0,Y 538.369,Z 208.021,A -85,B 0,C 180,E1 -3867.383,E2 -3867.383} C_VEL
LIN {X 0,Y 538.174,Z 223.393,A -85,B 0,C 180,E1 -3870.305,E2 -3870.305} C_VEL
LIN {X 0,Y 539.716,Z 231.876,A -85,B 0,C 180,E1 -3870.468,E2 -3870.468} C_VEL
LIN {X 0,Y 539.308,Z 330.055,A -85,B 0,C 180,E1 -3871.798,E2 -3871.798} C_VEL
LIN {X 0,Y 539.147,Z 343.092,A -85,B 0,C 180,E1 -3872.126,E2 -3872.126} C_VEL
LIN {X 0,Y 538.965,Z 356.173,A -85,B 0,C 180,E1 -3872.617,E2 -3872.617} C_VEL
LIN {X 0,Y 538.762,Z 367.209,A -85,B 0,C 180,E1 -3873.179,E2 -3873.179} C_VEL
LIN {X 0,Y 538.505,Z 378.679,A -85,B 0,C 180,E1 -3873.93,E2 -3873.93} C_VEL
LIN {X 0,Y 538.313,Z 389,A -85,B 0,C 180,E1 -3874.775,E2 -3874.775} C_VEL
LIN {X 0,Y 538.056,Z 397.495,A -85,B 0,C 180,E1 -3875.623,E2 -3875.623} C_VEL
LIN {X 0,Y 537.941,Z 405.335,A -85,B 0,C 180,E1 -3876.568,E2 -3876.568} C_VEL
LIN {X 0,Y 537.807,Z 412.981,A -85,B 0,C 180,E1 -3877.698,E2 -3877.698} C_VEL
LIN {X 0,Y 537.678,Z 420.054,A -85,B 0,C 180,E1 -3879.025,E2 -3879.025} C_VEL
LIN {X 0,Y 537.585,Z 424.778,A -85,B 0,C 180,E1 -3880.166,E2 -3880.166} C_VEL
LIN {X 0,Y 537.553,Z 428.413,A -85,B 0,C 180,E1 -3881.319,E2 -3881.319} C_VEL
LIN {X 0,Y 537.496,Z 430.247,A -85,B 0,C 180,E1 -3882.076,E2 -3882.076} C_VEL
LIN {X 0,Y 537.494,Z 431.628,A -85,B 0,C 180,E1 -3882.843,E2 -3882.843} C_VEL
LIN {X 0,Y 537.474,Z 432.609,A -85,B 0,C 180,E1 -3883.613,E2 -3883.613} C_VEL
LIN {X 0,Y 537.499,Z 433.266,A -85,B 0,C 180,E1 -3884.631,E2 -3884.631} C_VEL
LIN {X 0,Y 537.455,Z 433.046,A -85,B 0,C 180,E1 -3885.938,E2 -3885.938} C_VEL
LIN {X 0,Y 537.51,Z 431.469,A -85,B 0,C 180,E1 -3887.354,E2 -3887.354} C_VEL
LIN {X 0,Y 537.516,Z 428.668,A -85,B 0,C 180,E1 -3888.683,E2 -3888.683} C_VEL
LIN {X 0,Y 537.598,Z 424.99,A -85,B 0,C 180,E1 -3889.87,E2 -3889.87} C_VEL
LIN {X 0,Y 537.656,Z 420.061,A -85,B 0,C 180,E1 -3891.067,E2 -3891.067} C_VEL
LIN {X 0,Y 537.776,Z 413.71,A -85,B 0,C 180,E1 -3892.27,E2 -3892.27} C_VEL
LIN {X 0,Y 537.94,Z 405.662,A -85,B 0,C 180,E1 -3893.482,E2 -3893.482} C_VEL
LIN {X 0,Y 538.107,Z 397.222,A -85,B 0,C 180,E1 -3894.498,E2 -3894.498} C_VEL
LIN {X 0,Y 538.349,Z 386.754,A -85,B 0,C 180,E1 -3895.518,E2 -3895.518} C_VEL
LIN {X 0,Y 538.553,Z 376.262,A -85,B 0,C 180,E1 -3896.339,E2 -3896.339} C_VEL
LIN {X 0,Y 538.862,Z 364.615,A -85,B 0,C 180,E1 -3897.054,E2 -3897.054} C_VEL
LIN {X 0,Y 539.022,Z 352.399,A -85,B 0,C 180,E1 -3897.634,E2 -3897.634} C_VEL
LIN {X 0,Y 539.174,Z 339.878,A -85,B 0,C 180,E1 -3898.064,E2 -3898.064} C_VEL
LIN {X 0,Y 539.272,Z 326.794,A -85,B 0,C 180,E1 -3898.349,E2 -3898.349} C_VEL
LIN {X 0,Y 539.589,Z 231.153,A -85,B 0,C 180,E1 -3899.636,E2 -3899.636} C_VEL
LIN {X 0,Y 538.174,Z 223.213,A -85,B 0,C 180,E1 -3899.804,E2 -3899.804} C_VEL
LIN {X 0,Y 538.318,Z 209.599,A -85,B 0,C 180,E1 -3902.361,E2 -3902.361} C_VEL
LIN {X 0,Y 538.14,Z 202.654,A -85,B 0,C 180,E1 -3903.653,E2 -3903.653} C_VEL
LIN {X 0,Y 538.022,Z 202.466,A -85,B 0,C 180,E1 -3906.931,E2 -3906.931} C_VEL
LIN {X 0,Y 538.042,Z 202.463,A -85,B 0,C 180,E1 -3909.793,E2 -3909.793} C_VEL
LIN {X 0,Y 538.01,Z 202.467,A -85,B 0,C 180,E1 -3912.784,E2 -3912.784} C_VEL
LIN {X 0,Y 538.012,Z 202.469,A -85,B 0,C 180,E1 -3915.924,E2 -3915.924} C_VEL
LIN {X 0,Y 538.059,Z 202.458,A -85,B 0,C 180,E1 -3919.247,E2 -3919.247} C_VEL
LIN {X 0,Y 537.973,Z 202.475,A -85,B 0,C 180,E1 -3922.121,E2 -3922.121} C_VEL
LIN {X 0,Y 537.999,Z 202.464,A -85,B 0,C 180,E1 -3924.916,E2 -3924.916} C_VEL
LIN {X 0,Y 538.008,Z 202.468,A -85,B 0,C 180,E1 -3927.617,E2 -3927.617} C_VEL
LIN {X 0,Y 538.018,Z 202.465,A -85,B 0,C 180,E1 -3930.239,E2 -3930.239} C_VEL
LIN {X 0,Y 538.044,Z 202.458,A -85,B 0,C 180,E1 -3932.795,E2 -3932.795} C_VEL
LIN {X 0,Y 538.027,Z 202.461,A -85,B 0,C 180,E1 -3935.292,E2 -3935.292} C_VEL
LIN {X 0,Y 538.017,Z 202.465,A -85,B 0,C 180,E1 -3938.032,E2 -3938.032} C_VEL
LIN {X 0,Y 538.012,Z 202.463,A -85,B 0,C 180,E1 -3940.939,E2 -3940.939} C_VEL
LIN {X 0,Y 538.026,Z 202.464,A -85,B 0,C 180,E1 -3943.299,E2 -3943.299} C_VEL
LIN {X 0,Y 538.032,Z 202.468,A -85,B 0,C 180,E1 -3945.63,E2 -3945.63} C_VEL
LIN {X 0,Y 538.057,Z 202.457,A -85,B 0,C 180,E1 -3948.701,E2 -3948.701} C_VEL
LIN {X 0,Y 538.058,Z 202.46,A -85,B 0,C 180,E1 -3951.739,E2 -3951.739} C_VEL
LIN {X 0,Y 538.095,Z 202.453,A -85,B 0,C 180,E1 -3954.003,E2 -3954.003} C_VEL
LIN {X 0,Y 538.111,Z 202.452,A -85,B 0,C 180,E1 -3957.006,E2 -3957.006} C_VEL
LIN {X 0,Y 538.129,Z 202.447,A -85,B 0,C 180,E1 -3960,E2 -3960} C_VEL
LIN {X 0,Y 538.109,Z 202.455,A -85,B 0,C 180,E1 -3962.995,E2 -3962.995} C_VEL
LIN {X 0,Y 538.084,Z 202.451,A -85,B 0,C 180,E1 -3965.998,E2 -3965.998} C_VEL
LIN {X 0,Y 538.029,Z 202.468,A -85,B 0,C 180,E1 -3969.019,E2 -3969.019} C_VEL
LIN {X 0,Y 538.049,Z 202.457,A -85,B 0,C 180,E1 -3972.064,E2 -3972.064} C_VEL
LIN {X 0,Y 538.011,Z 202.468,A -85,B 0,C 180,E1 -3975.145,E2 -3975.145} C_VEL
LIN {X 0,Y 537.991,Z 202.466,A -85,B 0,C 180,E1 -3978.272,E2 -3978.272} C_VEL
LIN {X 0,Y 538.008,Z 202.469,A -85,B 0,C 180,E1 -3980.653,E2 -3980.653} C_VEL
LIN {X 0,Y 537.968,Z 202.467,A -85,B 0,C 180,E1 -3983.89,E2 -3983.89} C_VEL
LIN {X 0,Y 537.997,Z 202.47,A -85,B 0,C 180,E1 -3986.369,E2 -3986.369} C_VEL
LIN {X 0,Y 538.004,Z 202.469,A -85,B 0,C 180,E1 -3988.935,E2 -3988.935} C_VEL
LIN {X 0,Y 537.985,Z 202.467,A -85,B 0,C 180,E1 -3991.889,E2 -3991.889} C_VEL
LIN {X 0,Y 537.984,Z 202.474,A -85,B 0,C 180,E1 -3994.618,E2 -3994.618} C_VEL
LIN {X 0,Y 537.977,Z 202.467,A -85,B 0,C 180,E1 -3997.171,E2 -3997.171} C_VEL
LIN {X 0,Y 537.989,Z 202.468,A -85,B 0,C 180,E1 -3999.8,E2 -3999.8} C_VEL
LIN {X 0,Y 538.003,Z 202.467,A -85,B 0,C 180,E1 -4002.788,E2 -4002.788} C_VEL
LIN {X 0,Y 538.004,Z 202.468,A -85,B 0,C 180,E1 -4005.929,E2 -4005.929} C_VEL
LIN {X 0,Y 538.011,Z 202.463,A -85,B 0,C 180,E1 -4009.258,E2 -4009.258} C_VEL
LIN {X 0,Y 537.98,Z 202.475,A -85,B 0,C 180,E1 -4012.124,E2 -4012.124} C_VEL
LIN {X 0,Y 537.999,Z 202.466,A -85,B 0,C 180,E1 -4014.918,E2 -4014.918} C_VEL
LIN {X 0,Y 538.012,Z 202.468,A -85,B 0,C 180,E1 -4017.619,E2 -4017.619} C_VEL
LIN {X 0,Y 538.008,Z 202.47,A -85,B 0,C 180,E1 -4020.24,E2 -4020.24} C_VEL
LIN {X 0,Y 538.028,Z 202.464,A -85,B 0,C 180,E1 -4022.795,E2 -4022.795} C_VEL
LIN {X 0,Y 538.078,Z 202.586,A -85,B 0,C 180,E1 -4025.436,E2 -4025.436} C_VEL
LIN {X 0,Y 539.296,Z 209.912,A -85,B 0,C 180,E1 -4026.581,E2 -4026.581} C_VEL
LIN {X 0,Y 538.942,Z 231.09,A -85,B 0,C 180,E1 -4029.692,E2 -4029.692} C_VEL
LIN {X 0,Y 538.592,Z 252.075,A -85,B 0,C 180,E1 -4032.731,E2 -4032.731} C_VEL
LIN {X 0,Y 538.283,Z 269.773,A -85,B 0,C 180,E1 -4035.245,E2 -4035.245} C_VEL
LIN {X 0,Y 539.657,Z 279.273,A -85,B 0,C 180,E1 -4035.411,E2 -4035.411} C_VEL
LIN {X 0,Y 539.301,Z 378.093,A -85,B 0,C 180,E1 -4036.745,E2 -4036.745} C_VEL
LIN {X 0,Y 539.083,Z 391.425,A -85,B 0,C 180,E1 -4037.075,E2 -4037.075} C_VEL
LIN {X 0,Y 538.917,Z 403.634,A -85,B 0,C 180,E1 -4037.526,E2 -4037.526} C_VEL
LIN {X 0,Y 538.749,Z 415.289,A -85,B 0,C 180,E1 -4038.104,E2 -4038.104} C_VEL
LIN {X 0,Y 538.493,Z 426.295,A -85,B 0,C 180,E1 -4038.805,E2 -4038.805} C_VEL
LIN {X 0,Y 538.27,Z 436.998,A -85,B 0,C 180,E1 -4039.657,E2 -4039.657} C_VEL
LIN {X 0,Y 538.027,Z 446.644,A -85,B 0,C 180,E1 -4040.602,E2 -4040.602} C_VEL
LIN {X 0,Y 537.922,Z 454.557,A -85,B 0,C 180,E1 -4041.547,E2 -4041.547} C_VEL
LIN {X 0,Y 537.756,Z 462.284,A -85,B 0,C 180,E1 -4042.679,E2 -4042.679} C_VEL
LIN {X 0,Y 537.675,Z 469.409,A -85,B 0,C 180,E1 -4043.997,E2 -4043.997} C_VEL
LIN {X 0,Y 537.54,Z 474.146,A -85,B 0,C 180,E1 -4045.124,E2 -4045.124} C_VEL
LIN {X 0,Y 537.591,Z 477.772,A -85,B 0,C 180,E1 -4046.251,E2 -4046.251} C_VEL
LIN {X 0,Y 537.551,Z 479.64,A -85,B 0,C 180,E1 -4047.001,E2 -4047.001} C_VEL
LIN {X 0,Y 537.49,Z 481.039,A -85,B 0,C 180,E1 -4047.751,E2 -4047.751} C_VEL
LIN {X 0,Y 537.443,Z 482.648,A -85,B 0,C 180,E1 -4049.25,E2 -4049.25} C_VEL
LIN {X 0,Y 537.443,Z 482.867,A -85,B 0,C 180,E1 -4049.999,E2 -4049.999} C_VEL
LIN {X 0,Y 537.443,Z 482.651,A -85,B 0,C 180,E1 -4050.748,E2 -4050.748} C_VEL
LIN {X 0,Y 537.49,Z 481.047,A -85,B 0,C 180,E1 -4052.247,E2 -4052.247} C_VEL
LIN {X 0,Y 537.551,Z 479.651,A -85,B 0,C 180,E1 -4052.996,E2 -4052.996} C_VEL
LIN {X 0,Y 537.603,Z 476.709,A -85,B 0,C 180,E1 -4054.121,E2 -4054.121} C_VEL
LIN {X 0,Y 537.587,Z 472.723,A -85,B 0,C 180,E1 -4055.249,E2 -4055.249} C_VEL
LIN {X 0,Y 537.652,Z 466.619,A -85,B 0,C 180,E1 -4056.561,E2 -4056.561} C_VEL
LIN {X 0,Y 537.795,Z 459.903,A -85,B 0,C 180,E1 -4057.696,E2 -4057.696} C_VEL
LIN {X 0,Y 537.948,Z 451.597,A -85,B 0,C 180,E1 -4058.828,E2 -4058.828} C_VEL
LIN {X 0,Y 538.117,Z 443.087,A -85,B 0,C 180,E1 -4059.773,E2 -4059.773} C_VEL
LIN {X 0,Y 538.381,Z 432.577,A -85,B 0,C 180,E1 -4060.718,E2 -4060.718} C_VEL
LIN {X 0,Y 538.629,Z 421.145,A -85,B 0,C 180,E1 -4061.544,E2 -4061.544} C_VEL
LIN {X 0,Y 538.821,Z 410.789,A -85,B 0,C 180,E1 -4062.139,E2 -4062.139} C_VEL
LIN {X 0,Y 538.993,Z 399.11,A -85,B 0,C 180,E1 -4062.661,E2 -4062.661} C_VEL
LIN {X 0,Y 539.213,Z 386.581,A -85,B 0,C 180,E1 -4063.062,E2 -4063.062} C_VEL
LIN {X 0,Y 539.337,Z 373.917,A -85,B 0,C 180,E1 -4063.323,E2 -4063.323} C_VEL
LIN {X 0,Y 539.495,Z 277.51,A -85,B 0,C 180,E1 -4064.618,E2 -4064.618} C_VEL
LIN {X 0,Y 538.341,Z 269.558,A -85,B 0,C 180,E1 -4064.773,E2 -4064.773} C_VEL
LIN {X 0,Y 538.617,Z 249.047,A -85,B 0,C 180,E1 -4067.726,E2 -4067.726} C_VEL
LIN {X 0,Y 539.03,Z 227.886,A -85,B 0,C 180,E1 -4070.808,E2 -4070.808} C_VEL
LIN {X 0,Y 539.35,Z 210.281,A -85,B 0,C 180,E1 -4073.414,E2 -4073.414} C_VEL
LIN {X 0,Y 538.048,Z 202.464,A -85,B 0,C 180,E1 -4074.658,E2 -4074.658} C_VEL
LIN {X 0,Y 538.049,Z 202.461,A -85,B 0,C 180,E1 -4077.349,E2 -4077.349} C_VEL
LIN {X 0,Y 538.003,Z 202.47,A -85,B 0,C 180,E1 -4079.758,E2 -4079.758} C_VEL
LIN {X 0,Y 538.009,Z 202.467,A -85,B 0,C 180,E1 -4082.379,E2 -4082.379} C_VEL
LIN {X 0,Y 538,Z 202.464,A -85,B 0,C 180,E1 -4085.079,E2 -4085.079} C_VEL
LIN {X 0,Y 537.971,Z 202.476,A -85,B 0,C 180,E1 -4087.874,E2 -4087.874} C_VEL
LIN {X 0,Y 538.026,Z 202.461,A -85,B 0,C 180,E1 -4090.772,E2 -4090.772} C_VEL
LIN {X 0,Y 537.995,Z 202.471,A -85,B 0,C 180,E1 -4094.07,E2 -4094.07} C_VEL
LIN {X 0,Y 537.993,Z 202.467,A -85,B 0,C 180,E1 -4097.211,E2 -4097.211} C_VEL
LIN {X 0,Y 538.024,Z 202.464,A -85,B 0,C 180,E1 -4100.203,E2 -4100.203} C_VEL
LIN {X 0,Y 537.994,Z 202.466,A -85,B 0,C 180,E1 -4103.064,E2 -4103.064} C_VEL
LIN {X 0,Y 537.992,Z 202.472,A -85,B 0,C 180,E1 -4105.824,E2 -4105.824} C_VEL
LIN {X 0,Y 537.981,Z 202.466,A -85,B 0,C 180,E1 -4108.497,E2 -4108.497} C_VEL
LIN {X 0,Y 538.014,Z 202.465,A -85,B 0,C 180,E1 -4111.097,E2 -4111.097} C_VEL
LIN {X 0,Y 538.003,Z 202.471,A -85,B 0,C 180,E1 -4113.631,E2 -4113.631} C_VEL
LIN {X 0,Y 538.01,Z 202.464,A -85,B 0,C 180,E1 -4116.112,E2 -4116.112} C_VEL
LIN {X 0,Y 537.989,Z 202.465,A -85,B 0,C 180,E1 -4118.544,E2 -4118.544} C_VEL
LIN {X 0,Y 537.992,Z 202.468,A -85,B 0,C 180,E1 -4120.938,E2 -4120.938} C_VEL
LIN {X 0,Y 538.006,Z 202.472,A -85,B 0,C 180,E1 -4123.298,E2 -4123.298} C_VEL
LIN {X 0,Y 537.987,Z 202.466,A -85,B 0,C 180,E1 -4126.4,E2 -4126.4} C_VEL
LIN {X 0,Y 538.053,Z 202.459,A -85,B 0,C 180,E1 -4128.701,E2 -4128.701} C_VEL
LIN {X 0,Y 538.036,Z 202.462,A -85,B 0,C 180,E1 -4131.739,E2 -4131.739} C_VEL
LIN {X 0,Y 538.077,Z 202.455,A -85,B 0,C 180,E1 -4134.002,E2 -4134.002} C_VEL
LIN {X 0,Y 538.092,Z 202.46,A -85,B 0,C 180,E1 -4137.005,E2 -4137.005} C_VEL
LIN {X 0,Y 538.108,Z 202.451,A -85,B 0,C 180,E1 -4140,E2 -4140} C_VEL
LIN {X 0,Y 538.09,Z 202.462,A -85,B 0,C 180,E1 -4142.994,E2 -4142.994} C_VEL
LIN {X 0,Y 538.063,Z 202.456,A -85,B 0,C 180,E1 -4145.998,E2 -4145.998} C_VEL
LIN {X 0,Y 538.021,Z 202.469,A -85,B 0,C 180,E1 -4149.018,E2 -4149.018} C_VEL
LIN {X 0,Y 538.027,Z 202.461,A -85,B 0,C 180,E1 -4152.064,E2 -4152.064} C_VEL
LIN {X 0,Y 537.99,Z 202.47,A -85,B 0,C 180,E1 -4155.145,E2 -4155.145} C_VEL
LIN {X 0,Y 538.038,Z 202.46,A -85,B 0,C 180,E1 -4157.554,E2 -4157.554} C_VEL
LIN {X 0,Y 537.99,Z 202.474,A -85,B 0,C 180,E1 -4160.653,E2 -4160.653} C_VEL
LIN {X 0,Y 537.99,Z 202.466,A -85,B 0,C 180,E1 -4163.889,E2 -4163.889} C_VEL
LIN {X 0,Y 537.999,Z 202.47,A -85,B 0,C 180,E1 -4166.369,E2 -4166.369} C_VEL
LIN {X 0,Y 537.988,Z 202.47,A -85,B 0,C 180,E1 -4168.937,E2 -4168.937} C_VEL
LIN {X 0,Y 537.982,Z 202.468,A -85,B 0,C 180,E1 -4171.893,E2 -4171.893} C_VEL
LIN {X 0,Y 537.987,Z 202.473,A -85,B 0,C 180,E1 -4174.624,E2 -4174.624} C_VEL
LIN {X 0,Y 537.968,Z 202.469,A -85,B 0,C 180,E1 -4177.174,E2 -4177.174} C_VEL
LIN {X 0,Y 537.984,Z 202.466,A -85,B 0,C 180,E1 -4180.294,E2 -4180.294} C_VEL
LIN {X 0,Y 537.339,Z 202.55,A -85,B 0,C 180,E1 -4180.919,E2 -4180.919} C_VEL
LIN {X 0,Y 534.489,Z 202.905,A -85,B 0,C 180,E1 -4181.934,E2 -4181.934} C_VEL
LIN {X 0,Y 532.062,Z 203.207,A -85,B 0,C 180,E1 -4182.751,E2 -4182.751} C_VEL
LIN {X 0,Y 531.013,Z 203.335,A -85,B 0,C 180,E1 -4183.383,E2 -4183.383} C_VEL
LIN {X 0,Y 530.924,Z 203.346,A -85,B 0,C 180,E1 -4183.596,E2 -4183.596} C_VEL
LIN {X 0,Y 530.925,Z 203.351,A -85,B 0,C 180,E1 -4186.508,E2 -4186.508} C_VEL
LIN {X 0,Y 530.959,Z 203.342,A -85,B 0,C 180,E1 -4188.979,E2 -4188.979} C_VEL
LIN {X 0,Y 530.929,Z 203.346,A -85,B 0,C 180,E1 -4191.533,E2 -4191.533} C_VEL
LIN {X 0,Y 530.954,Z 203.347,A -85,B 0,C 180,E1 -4194.385,E2 -4194.385} C_VEL
LIN {X 0,Y 530.945,Z 203.343,A -85,B 0,C 180,E1 -4197.137,E2 -4197.137} C_VEL
LIN {X 0,Y 530.95,Z 203.348,A -85,B 0,C 180,E1 -4199.806,E2 -4199.806} C_VEL
LIN {X 0,Y 530.994,Z 203.34,A -85,B 0,C 180,E1 -4202.471,E2 -4202.471} C_VEL
LIN {X 0,Y 530.98,Z 203.339,A -85,B 0,C 180,E1 -4204.945,E2 -4204.945} C_VEL
LIN {X 0,Y 530.959,Z 203.345,A -85,B 0,C 180,E1 -4208.25,E2 -4208.25} C_VEL
LIN {X 0,Y 530.971,Z 203.34,A -85,B 0,C 180,E1 -4210.68,E2 -4210.68} C_VEL
LIN {X 0,Y 530.951,Z 203.343,A -85,B 0,C 180,E1 -4213.073,E2 -4213.073} C_VEL
LIN {X 0,Y 531.001,Z 203.34,A -85,B 0,C 180,E1 -4215.438,E2 -4215.438} C_VEL
LIN {X 0,Y 531.029,Z 203.333,A -85,B 0,C 180,E1 -4218.552,E2 -4218.552} C_VEL
LIN {X 0,Y 531.047,Z 203.339,A -85,B 0,C 180,E1 -4221.631,E2 -4221.631} C_VEL
LIN {X 0,Y 531.111,Z 203.325,A -85,B 0,C 180,E1 -4224.687,E2 -4224.687} C_VEL
LIN {X 0,Y 530.961,Z 203.438,A -85,B 0,C 180,E1 -4226.231,E2 -4226.231} C_VEL
LIN {X 0,Y 531.378,Z 207.205,A -85,B 0,C 180,E1 -4226.969,E2 -4226.969} C_VEL
LIN {X 0,Y 531.22,Z 221.102,A -85,B 0,C 180,E1 -4229.622,E2 -4229.622} C_VEL
LIN {X 0,Y 531.186,Z 223.589,A -85,B 0,C 180,E1 -4230.096,E2 -4230.096} C_VEL
LIN {X 0,Y 532.856,Z 232.83,A -85,B 0,C 180,E1 -4230.285,E2 -4230.285} C_VEL
LIN {X 0,Y 532.423,Z 330.733,A -85,B 0,C 180,E1 -4231.632,E2 -4231.632} C_VEL
LIN {X 0,Y 532.249,Z 342.913,A -85,B 0,C 180,E1 -4231.94,E2 -4231.94} C_VEL
LIN {X 0,Y 532.076,Z 355.559,A -85,B 0,C 180,E1 -4232.414,E2 -4232.414} C_VEL
LIN {X 0,Y 531.826,Z 367.659,A -85,B 0,C 180,E1 -4233.031,E2 -4233.031} C_VEL
LIN {X 0,Y 531.538,Z 379.111,A -85,B 0,C 180,E1 -4233.792,E2 -4233.792} C_VEL
LIN {X 0,Y 531.324,Z 389.415,A -85,B 0,C 180,E1 -4234.648,E2 -4234.648} C_VEL
LIN {X 0,Y 531.046,Z 397.896,A -85,B 0,C 180,E1 -4235.507,E2 -4235.507} C_VEL
LIN {X 0,Y 530.896,Z 406.673,A -85,B 0,C 180,E1 -4236.595,E2 -4236.595} C_VEL
LIN {X 0,Y 530.75,Z 414.463,A -85,B 0,C 180,E1 -4237.801,E2 -4237.801} C_VEL
LIN {X 0,Y 530.598,Z 421.305,A -85,B 0,C 180,E1 -4239.146,E2 -4239.146} C_VEL
LIN {X 0,Y 530.509,Z 425.819,A -85,B 0,C 180,E1 -4240.303,E2 -4240.303} C_VEL
LIN {X 0,Y 530.477,Z 429.249,A -85,B 0,C 180,E1 -4241.463,E2 -4241.463} C_VEL
LIN {X 0,Y 530.402,Z 430.958,A -85,B 0,C 180,E1 -4242.24,E2 -4242.24} C_VEL
LIN {X 0,Y 530.393,Z 432.252,A -85,B 0,C 180,E1 -4243.018,E2 -4243.018} C_VEL
LIN {X 0,Y 530.402,Z 433.145,A -85,B 0,C 180,E1 -4243.798,E2 -4243.798} C_VEL
LIN {X 0,Y 530.414,Z 433.608,A -85,B 0,C 180,E1 -4244.705,E2 -4244.705} C_VEL
LIN {X 0,Y 530.361,Z 433.244,A -85,B 0,C 180,E1 -4246.157,E2 -4246.157} C_VEL
LIN {X 0,Y 530.41,Z 431.709,A -85,B 0,C 180,E1 -4247.445,E2 -4247.445} C_VEL
LIN {X 0,Y 530.448,Z 428.414,A -85,B 0,C 180,E1 -4248.941,E2 -4248.941} C_VEL
LIN {X 0,Y 530.526,Z 424.535,A -85,B 0,C 180,E1 -4250.146,E2 -4250.146} C_VEL
LIN {X 0,Y 530.608,Z 419.388,A -85,B 0,C 180,E1 -4251.36,E2 -4251.36} C_VEL
LIN {X 0,Y 530.763,Z 412.79,A -85,B 0,C 180,E1 -4252.581,E2 -4252.581} C_VEL
LIN {X 0,Y 530.938,Z 404.712,A -85,B 0,C 180,E1 -4253.76,E2 -4253.76} C_VEL
LIN {X 0,Y 531.137,Z 395.542,A -85,B 0,C 180,E1 -4254.841,E2 -4254.841} C_VEL
LIN {X 0,Y 531.368,Z 385.778,A -85,B 0,C 180,E1 -4255.772,E2 -4255.772} C_VEL
LIN {X 0,Y 531.64,Z 375.054,A -85,B 0,C 180,E1 -4256.591,E2 -4256.591} C_VEL
LIN {X 0,Y 531.948,Z 362.826,A -85,B 0,C 180,E1 -4257.328,E2 -4257.328} C_VEL
LIN {X 0,Y 532.147,Z 350.728,A -85,B 0,C 180,E1 -4257.88,E2 -4257.88} C_VEL
LIN {X 0,Y 532.312,Z 337.4,A -85,B 0,C 180,E1 -4258.308,E2 -4258.308} C_VEL
LIN {X 0,Y 532.397,Z 324.822,A -85,B 0,C 180,E1 -4258.561,E2 -4258.561} C_VEL
LIN {X 0,Y 532.776,Z 232.267,A -85,B 0,C 180,E1 -4259.816,E2 -4259.816} C_VEL
LIN {X 0,Y 531.196,Z 223.558,A -85,B 0,C 180,E1 -4259.997,E2 -4259.997} C_VEL
LIN {X 0,Y 531.353,Z 208.366,A -85,B 0,C 180,E1 -4262.838,E2 -4262.838} C_VEL
LIN {X 0,Y 531.044,Z 203.338,A -85,B 0,C 180,E1 -4263.795,E2 -4263.795} C_VEL
LIN {X 0,Y 530.96,Z 203.35,A -85,B 0,C 180,E1 -4266.556,E2 -4266.556} C_VEL
LIN {X 0,Y 530.994,Z 203.342,A -85,B 0,C 180,E1 -4269.856,E2 -4269.856} C_VEL
LIN {X 0,Y 530.973,Z 203.349,A -85,B 0,C 180,E1 -4272.454,E2 -4272.454} C_VEL
LIN {X 0,Y 530.971,Z 203.343,A -85,B 0,C 180,E1 -4275.619,E2 -4275.619} C_VEL
LIN {X 0,Y 530.989,Z 203.342,A -85,B 0,C 180,E1 -4278.564,E2 -4278.564} C_VEL
LIN {X 0,Y 530.948,Z 203.344,A -85,B 0,C 180,E1 -4281.344,E2 -4281.344} C_VEL
LIN {X 0,Y 530.96,Z 203.344,A -85,B 0,C 180,E1 -4284.381,E2 -4284.381} C_VEL
LIN {X 0,Y 530.951,Z 203.343,A -85,B 0,C 180,E1 -4287.133,E2 -4287.133} C_VEL
LIN {X 0,Y 530.961,Z 203.348,A -85,B 0,C 180,E1 -4289.803,E2 -4289.803} C_VEL
LIN {X 0,Y 530.991,Z 203.338,A -85,B 0,C 180,E1 -4292.465,E2 -4292.465} C_VEL
LIN {X 0,Y 530.982,Z 203.337,A -85,B 0,C 180,E1 -4294.942,E2 -4294.942} C_VEL
LIN {X 0,Y 530.978,Z 203.344,A -85,B 0,C 180,E1 -4297.889,E2 -4297.889} C_VEL
LIN {X 0,Y 530.968,Z 203.34,A -85,B 0,C 180,E1 -4300.677,E2 -4300.677} C_VEL
LIN {X 0,Y 530.987,Z 203.338,A -85,B 0,C 180,E1 -4303.071,E2 -4303.071} C_VEL
LIN {X 0,Y 531.008,Z 203.343,A -85,B 0,C 180,E1 -4305.436,E2 -4305.436} C_VEL
LIN {X 0,Y 531.013,Z 203.334,A -85,B 0,C 180,E1 -4308.549,E2 -4308.549} C_VEL
LIN {X 0,Y 531.027,Z 203.337,A -85,B 0,C 180,E1 -4311.629,E2 -4311.629} C_VEL
LIN {X 0,Y 531.054,Z 203.331,A -85,B 0,C 180,E1 -4313.923,E2 -4313.923} C_VEL
LIN {X 0,Y 531.077,Z 203.328,A -85,B 0,C 180,E1 -4316.966,E2 -4316.966} C_VEL
LIN {X 0,Y 531.101,Z 203.322,A -85,B 0,C 180,E1 -4320,E2 -4320} C_VEL
LIN {X 0,Y 531.075,Z 203.332,A -85,B 0,C 180,E1 -4323.035,E2 -4323.035} C_VEL
LIN {X 0,Y 531.04,Z 203.328,A -85,B 0,C 180,E1 -4326.078,E2 -4326.078} C_VEL
LIN {X 0,Y 530.993,Z 203.342,A -85,B 0,C 180,E1 -4329.139,E2 -4329.139} C_VEL
LIN {X 0,Y 531.033,Z 203.332,A -85,B 0,C 180,E1 -4331.681,E2 -4331.681} C_VEL
LIN {X 0,Y 530.998,Z 203.342,A -85,B 0,C 180,E1 -4334.956,E2 -4334.956} C_VEL
LIN {X 0,Y 530.949,Z 203.342,A -85,B 0,C 180,E1 -4337.725,E2 -4337.725} C_VEL
LIN {X 0,Y 530.995,Z 203.337,A -85,B 0,C 180,E1 -4340.129,E2 -4340.129} C_VEL
LIN {X 0,Y 530.912,Z 203.354,A -85,B 0,C 180,E1 -4342.575,E2 -4342.575} C_VEL
LIN {X 0,Y 530.922,Z 203.35,A -85,B 0,C 180,E1 -4345.062,E2 -4345.062} C_VEL
LIN {X 0,Y 530.943,Z 203.342,A -85,B 0,C 180,E1 -4347.6,E2 -4347.6} C_VEL
LIN {X 0,Y 530.933,Z 203.348,A -85,B 0,C 180,E1 -4350.2,E2 -4350.2} C_VEL
LIN {X 0,Y 530.943,Z 203.348,A -85,B 0,C 180,E1 -4352.869,E2 -4352.869} C_VEL
LIN {X 0,Y 530.927,Z 203.346,A -85,B 0,C 180,E1 -4355.622,E2 -4355.622} C_VEL
LIN {X 0,Y 530.942,Z 203.35,A -85,B 0,C 180,E1 -4358.655,E2 -4358.655} C_VEL
LIN {X 0,Y 530.979,Z 203.336,A -85,B 0,C 180,E1 -4361.437,E2 -4361.437} C_VEL
LIN {X 0,Y 530.958,Z 203.347,A -85,B 0,C 180,E1 -4364.55,E2 -4364.55} C_VEL
LIN {X 0,Y 530.956,Z 203.346,A -85,B 0,C 180,E1 -4367.838,E2 -4367.838} C_VEL
LIN {X 0,Y 530.96,Z 203.345,A -85,B 0,C 180,E1 -4370.557,E2 -4370.557} C_VEL
LIN {X 0,Y 530.95,Z 203.343,A -85,B 0,C 180,E1 -4373.443,E2 -4373.443} C_VEL
LIN {X 0,Y 530.993,Z 203.341,A -85,B 0,C 180,E1 -4376.496,E2 -4376.496} C_VEL
LIN {X 0,Y 530.97,Z 203.343,A -85,B 0,C 180,E1 -4379.356,E2 -4379.356} C_VEL
LIN {X 0,Y 530.962,Z 203.347,A -85,B 0,C 180,E1 -4381.544,E2 -4381.544} C_VEL
LIN {X 0,Y 530.982,Z 203.347,A -85,B 0,C 180,E1 -4384.164,E2 -4384.164} C_VEL
LIN {X 0,Y 531.037,Z 203.359,A -85,B 0,C 180,E1 -4385.259,E2 -4385.259} C_VEL
LIN {X 0,Y 532.341,Z 210.931,A -85,B 0,C 180,E1 -4386.463,E2 -4386.463} C_VEL
LIN {X 0,Y 531.995,Z 230.021,A -85,B 0,C 180,E1 -4389.309,E2 -4389.309} C_VEL
LIN {X 0,Y 531.586,Z 251.727,A -85,B 0,C 180,E1 -4392.496,E2 -4392.496} C_VEL
LIN {X 0,Y 531.261,Z 269.314,A -85,B 0,C 180,E1 -4395.044,E2 -4395.044} C_VEL
LIN {X 0,Y 532.803,Z 280.138,A -85,B 0,C 180,E1 -4395.235,E2 -4395.235} C_VEL
LIN {X 0,Y 532.398,Z 377.713,A -85,B 0,C 180,E1 -4396.57,E2 -4396.57} C_VEL
LIN {X 0,Y 532.175,Z 391.06,A -85,B 0,C 180,E1 -4396.905,E2 -4396.905} C_VEL
LIN {X 0,Y 531.952,Z 404.404,A -85,B 0,C 180,E1 -4397.409,E2 -4397.409} C_VEL
LIN {X 0,Y 531.74,Z 416.3,A -85,B 0,C 180,E1 -4398.027,E2 -4398.027} C_VEL
LIN {X 0,Y 531.441,Z 428.543,A -85,B 0,C 180,E1 -4398.848,E2 -4398.848} C_VEL
LIN {X 0,Y 531.146,Z 438.777,A -85,B 0,C 180,E1 -4399.71,E2 -4399.71} C_VEL
LIN {X 0,Y 530.951,Z 447.988,A -85,B 0,C 180,E1 -4400.668,E2 -4400.668} C_VEL
LIN {X 0,Y 530.772,Z 456.966,A -85,B 0,C 180,E1 -4401.816,E2 -4401.816} C_VEL
LIN {X 0,Y 530.627,Z 464.193,A -85,B 0,C 180,E1 -4402.962,E2 -4402.962} C_VEL
LIN {X 0,Y 530.572,Z 470.779,A -85,B 0,C 180,E1 -4404.298,E2 -4404.298} C_VEL
LIN {X 0,Y 530.452,Z 475.132,A -85,B 0,C 180,E1 -4405.44,E2 -4405.44} C_VEL
LIN {X 0,Y 530.516,Z 477.442,A -85,B 0,C 180,E1 -4406.201,E2 -4406.201} C_VEL
LIN {X 0,Y 530.457,Z 479.31,A -85,B 0,C 180,E1 -4406.961,E2 -4406.961} C_VEL
LIN {X 0,Y 530.411,Z 480.711,A -85,B 0,C 180,E1 -4407.721,E2 -4407.721} C_VEL
LIN {X 0,Y 530.35,Z 482.321,A -85,B 0,C 180,E1 -4409.239,E2 -4409.239} C_VEL
LIN {X 0,Y 530.351,Z 482.54,A -85,B 0,C 180,E1 -4409.999,E2 -4409.999} C_VEL
LIN {X 0,Y 530.361,Z 481.717,A -85,B 0,C 180,E1 -4411.517,E2 -4411.517} C_VEL
LIN {X 0,Y 530.411,Z 480.722,A -85,B 0,C 180,E1 -4412.277,E2 -4412.277} C_VEL
LIN {X 0,Y 530.457,Z 479.325,A -85,B 0,C 180,E1 -4413.036,E2 -4413.036} C_VEL
LIN {X 0,Y 530.522,Z 476.384,A -85,B 0,C 180,E1 -4414.177,E2 -4414.177} C_VEL
LIN {X 0,Y 530.521,Z 472.397,A -85,B 0,C 180,E1 -4415.319,E2 -4415.319} C_VEL
LIN {X 0,Y 530.554,Z 466.876,A -85,B 0,C 180,E1 -4416.54,E2 -4416.54} C_VEL
LIN {X 0,Y 530.717,Z 459.573,A -85,B 0,C 180,E1 -4417.799,E2 -4417.799} C_VEL
LIN {X 0,Y 530.894,Z 451.267,A -85,B 0,C 180,E1 -4418.946,E2 -4418.946} C_VEL
LIN {X 0,Y 531.069,Z 442.755,A -85,B 0,C 180,E1 -4419.904,E2 -4419.904} C_VEL
LIN {X 0,Y 531.343,Z 432.242,A -85,B 0,C 180,E1 -4420.862,E2 -4420.862} C_VEL
LIN {X 0,Y 531.613,Z 421.37,A -85,B 0,C 180,E1 -4421.661,E2 -4421.661} C_VEL
LIN {X 0,Y 531.856,Z 410.45,A -85,B 0,C 180,E1 -4422.3,E2 -4422.3} C_VEL
LIN {X 0,Y 532.059,Z 398.765,A -85,B 0,C 180,E1 -4422.829,E2 -4422.829} C_VEL
LIN {X 0,Y 532.3,Z 386.227,A -85,B 0,C 180,E1 -4423.235,E2 -4423.235} C_VEL
LIN {X 0,Y 532.425,Z 373.543,A -85,B 0,C 180,E1 -4423.499,E2 -4423.499} C_VEL
LIN {X 0,Y 532.635,Z 278.398,A -85,B 0,C 180,E1 -4424.794,E2 -4424.794} C_VEL
LIN {X 0,Y 531.302,Z 269.306,A -85,B 0,C 180,E1 -4424.962,E2 -4424.962} C_VEL
LIN {X 0,Y 531.655,Z 247.726,A -85,B 0,C 180,E1 -4428.112,E2 -4428.112} C_VEL
LIN {X 0,Y 532.055,Z 227.573,A -85,B 0,C 180,E1 -4431.094,E2 -4431.094} C_VEL
LIN {X 0,Y 532.41,Z 211.327,A -85,B 0,C 180,E1 -4433.531,E2 -4433.531} C_VEL
LIN {X 0,Y 531.017,Z 203.339,A -85,B 0,C 180,E1 -4434.844,E2 -4434.844} C_VEL
LIN {X 0,Y 531.004,Z 203.341,A -85,B 0,C 180,E1 -4437.592,E2 -4437.592} C_VEL
LIN {X 0,Y 530.958,Z 203.343,A -85,B 0,C 180,E1 -4440.641,E2 -4440.641} C_VEL
LIN {X 0,Y 530.974,Z 203.344,A -85,B 0,C 180,E1 -4443.769,E2 -4443.769} C_VEL
LIN {X 0,Y 530.946,Z 203.344,A -85,B 0,C 180,E1 -4446.554,E2 -4446.554} C_VEL
LIN {X 0,Y 530.959,Z 203.349,A -85,B 0,C 180,E1 -4449.851,E2 -4449.851} C_VEL
LIN {X 0,Y 530.953,Z 203.344,A -85,B 0,C 180,E1 -4452.453,E2 -4452.453} C_VEL
LIN {X 0,Y 530.957,Z 203.347,A -85,B 0,C 180,E1 -4455.617,E2 -4455.617} C_VEL
LIN {X 0,Y 530.987,Z 203.338,A -85,B 0,C 180,E1 -4458.563,E2 -4458.563} C_VEL
LIN {X 0,Y 530.934,Z 203.348,A -85,B 0,C 180,E1 -4461.342,E2 -4461.342} C_VEL
LIN {X 0,Y 530.943,Z 203.344,A -85,B 0,C 180,E1 -4464.379,E2 -4464.379} C_VEL
LIN {X 0,Y 530.934,Z 203.347,A -85,B 0,C 180,E1 -4467.131,E2 -4467.131} C_VEL
LIN {X 0,Y 530.943,Z 203.349,A -85,B 0,C 180,E1 -4469.801,E2 -4469.801} C_VEL
LIN {X 0,Y 530.972,Z 203.339,A -85,B 0,C 180,E1 -4472.463,E2 -4472.463} C_VEL
LIN {X 0,Y 530.962,Z 203.343,A -85,B 0,C 180,E1 -4474.94,E2 -4474.94} C_VEL
LIN {X 0,Y 530.958,Z 203.344,A -85,B 0,C 180,E1 -4477.887,E2 -4477.887} C_VEL
LIN {X 0,Y 530.947,Z 203.343,A -85,B 0,C 180,E1 -4480.675,E2 -4480.675} C_VEL
LIN {X 0,Y 530.966,Z 203.345,A -85,B 0,C 180,E1 -4483.07,E2 -4483.07} C_VEL
LIN {X 0,Y 530.987,Z 203.345,A -85,B 0,C 180,E1 -4485.435,E2 -4485.435} C_VEL
LIN {X 0,Y 531.005,Z 203.336,A -85,B 0,C 180,E1 -4488.549,E2 -4488.549} C_VEL
LIN {X 0,Y 531.006,Z 203.339,A -85,B 0,C 180,E1 -4491.628,E2 -4491.628} C_VEL
LIN {X 0,Y 531.035,Z 203.332,A -85,B 0,C 180,E1 -4493.922,E2 -4493.922} C_VEL
LIN {X 0,Y 531.058,Z 203.336,A -85,B 0,C 180,E1 -4496.965,E2 -4496.965} C_VEL
LIN {X 0,Y 531.08,Z 203.326,A -85,B 0,C 180,E1 -4500,E2 -4500} C_VEL
LIN {X 0,Y 531.056,Z 203.338,A -85,B 0,C 180,E1 -4503.034,E2 -4503.034} C_VEL
LIN {X 0,Y 531.019,Z 203.334,A -85,B 0,C 180,E1 -4506.078,E2 -4506.078} C_VEL
LIN {X 0,Y 530.982,Z 203.344,A -85,B 0,C 180,E1 -4509.139,E2 -4509.139} C_VEL
LIN {X 0,Y 531.01,Z 203.335,A -85,B 0,C 180,E1 -4511.681,E2 -4511.681} C_VEL
LIN {X 0,Y 530.973,Z 203.347,A -85,B 0,C 180,E1 -4514.957,E2 -4514.957} C_VEL
LIN {X 0,Y 530.975,Z 203.339,A -85,B 0,C 180,E1 -4517.724,E2 -4517.724} C_VEL
LIN {X 0,Y 530.952,Z 203.348,A -85,B 0,C 180,E1 -4520.94,E2 -4520.94} C_VEL
LIN {X 0,Y 530.956,Z 203.343,A -85,B 0,C 180,E1 -4524.047,E2 -4524.047} C_VEL
LIN {X 0,Y 530.961,Z 203.348,A -85,B 0,C 180,E1 -4526.746,E2 -4526.746} C_VEL
LIN {X 0,Y 530.936,Z 203.344,A -85,B 0,C 180,E1 -4529.325,E2 -4529.325} C_VEL
LIN {X 0,Y 530.934,Z 203.347,A -85,B 0,C 180,E1 -4532.106,E2 -4532.106} C_VEL
LIN {X 0,Y 530.945,Z 203.347,A -85,B 0,C 180,E1 -4534.857,E2 -4534.857} C_VEL
LIN {X 0,Y 530.926,Z 203.345,A -85,B 0,C 180,E1 -4537.511,E2 -4537.511} C_VEL
LIN {X 0,Y 530.947,Z 203.351,A -85,B 0,C 180,E1 -4540.436,E2 -4540.436} C_VEL
LIN {X 0,Y 530.93,Z 203.345,A -85,B 0,C 180,E1 -4543.285,E2 -4543.285} C_VEL
LIN {X 0,Y 530.924,Z 203.346,A -85,B 0,C 180,E1 -4543.596,E2 -4543.596} C_VEL
LIN {X 0,Y 530.25,Z 203.437,A -85,B 0,C 180,E1 -4544.23,E2 -4544.23} C_VEL
LIN {X 0,Y 527.4,Z 203.79,A -85,B 0,C 180,E1 -4545.259,E2 -4545.259} C_VEL
LIN {X 0,Y 524.997,Z 204.09,A -85,B 0,C 180,E1 -4546.087,E2 -4546.087} C_VEL
LIN {X 0,Y 523.967,Z 204.215,A -85,B 0,C 180,E1 -4546.727,E2 -4546.727} C_VEL
LIN {X 0,Y 523.884,Z 204.223,A -85,B 0,C 180,E1 -4546.944,E2 -4546.944} C_VEL
LIN {X 0,Y 523.92,Z 204.223,A -85,B 0,C 180,E1 -4549.924,E2 -4549.924} C_VEL
LIN {X 0,Y 523.885,Z 204.223,A -85,B 0,C 180,E1 -4552.872,E2 -4552.872} C_VEL
LIN {X 0,Y 523.917,Z 204.222,A -85,B 0,C 180,E1 -4555.714,E2 -4555.714} C_VEL
LIN {X 0,Y 523.9,Z 204.224,A -85,B 0,C 180,E1 -4558.459,E2 -4558.459} C_VEL
LIN {X 0,Y 523.917,Z 204.218,A -85,B 0,C 180,E1 -4561.128,E2 -4561.128} C_VEL
LIN {X 0,Y 523.968,Z 204.222,A -85,B 0,C 180,E1 -4563.984,E2 -4563.984} C_VEL
LIN {X 0,Y 523.897,Z 204.221,A -85,B 0,C 180,E1 -4567.109,E2 -4567.109} C_VEL
LIN {X 0,Y 523.968,Z 204.221,A -85,B 0,C 180,E1 -4569.869,E2 -4569.869} C_VEL
LIN {X 0,Y 523.931,Z 204.217,A -85,B 0,C 180,E1 -4572.839,E2 -4572.839} C_VEL
LIN {X 0,Y 523.96,Z 204.215,A -85,B 0,C 180,E1 -4575.238,E2 -4575.238} C_VEL
LIN {X 0,Y 524.008,Z 204.208,A -85,B 0,C 180,E1 -4578.396,E2 -4578.396} C_VEL
LIN {X 0,Y 523.995,Z 204.215,A -85,B 0,C 180,E1 -4581.518,E2 -4581.518} C_VEL
LIN {X 0,Y 524.072,Z 204.202,A -85,B 0,C 180,E1 -4584.615,E2 -4584.615} C_VEL
LIN {X 0,Y 523.924,Z 204.346,A -85,B 0,C 180,E1 -4586.132,E2 -4586.132} C_VEL
LIN {X 0,Y 524.383,Z 209.387,A -85,B 0,C 180,E1 -4587.121,E2 -4587.121} C_VEL
LIN {X 0,Y 524.212,Z 223.912,A -85,B 0,C 180,E1 -4589.905,E2 -4589.905} C_VEL
LIN {X 0,Y 526.017,Z 233.771,A -85,B 0,C 180,E1 -4590.097,E2 -4590.097} C_VEL
LIN {X 0,Y 525.533,Z 330.314,A -85,B 0,C 180,E1 -4591.438,E2 -4591.438} C_VEL
LIN {X 0,Y 525.366,Z 342.726,A -85,B 0,C 180,E1 -4591.75,E2 -4591.75} C_VEL
LIN {X 0,Y 525.187,Z 354.947,A -85,B 0,C 180,E1 -4592.206,E2 -4592.206} C_VEL
LIN {X 0,Y 524.943,Z 366.447,A -85,B 0,C 180,E1 -4592.783,E2 -4592.783} C_VEL
LIN {X 0,Y 524.63,Z 376.98,A -85,B 0,C 180,E1 -4593.457,E2 -4593.457} C_VEL
LIN {X 0,Y 524.335,Z 387.737,A -85,B 0,C 180,E1 -4594.325,E2 -4594.325} C_VEL
LIN {X 0,Y 524.137,Z 396.516,A -85,B 0,C 180,E1 -4595.194,E2 -4595.194} C_VEL
LIN {X 0,Y 523.926,Z 404.611,A -85,B 0,C 180,E1 -4596.161,E2 -4596.161} C_VEL
LIN {X 0,Y 523.756,Z 412.567,A -85,B 0,C 180,E1 -4597.324,E2 -4597.324} C_VEL
LIN {X 0,Y 523.594,Z 418.972,A -85,B 0,C 180,E1 -4598.491,E2 -4598.491} C_VEL
LIN {X 0,Y 523.482,Z 424.059,A -85,B 0,C 180,E1 -4599.661,E2 -4599.661} C_VEL
LIN {X 0,Y 523.409,Z 428.013,A -85,B 0,C 180,E1 -4600.835,E2 -4600.835} C_VEL
LIN {X 0,Y 523.383,Z 430.046,A -85,B 0,C 180,E1 -4601.62,E2 -4601.62} C_VEL
LIN {X 0,Y 523.305,Z 431.668,A -85,B 0,C 180,E1 -4602.409,E2 -4602.409} C_VEL
LIN {X 0,Y 523.298,Z 432.869,A -85,B 0,C 180,E1 -4603.198,E2 -4603.198} C_VEL
LIN {X 0,Y 523.32,Z 433.609,A -85,B 0,C 180,E1 -4603.989,E2 -4603.989} C_VEL
LIN {X 0,Y 523.336,Z 433.951,A -85,B 0,C 180,E1 -4604.783,E2 -4604.783} C_VEL
LIN {X 0,Y 523.271,Z 433.9,A -85,B 0,C 180,E1 -4605.582,E2 -4605.582} C_VEL
LIN {X 0,Y 523.271,Z 433.403,A -85,B 0,C 180,E1 -4606.382,E2 -4606.382} C_VEL
LIN {X 0,Y 523.322,Z 431.932,A -85,B 0,C 180,E1 -4607.542,E2 -4607.542} C_VEL
LIN {X 0,Y 523.411,Z 428.162,A -85,B 0,C 180,E1 -4609.206,E2 -4609.206} C_VEL
LIN {X 0,Y 523.479,Z 424.081,A -85,B 0,C 180,E1 -4610.43,E2 -4610.43} C_VEL
LIN {X 0,Y 523.565,Z 418.689,A -85,B 0,C 180,E1 -4611.662,E2 -4611.662} C_VEL
LIN {X 0,Y 523.756,Z 411.755,A -85,B 0,C 180,E1 -4612.9,E2 -4612.9} C_VEL
LIN {X 0,Y 523.926,Z 404.33,A -85,B 0,C 180,E1 -4613.971,E2 -4613.971} C_VEL
LIN {X 0,Y 524.172,Z 394.802,A -85,B 0,C 180,E1 -4615.088,E2 -4615.088} C_VEL
LIN {X 0,Y 524.478,Z 384.663,A -85,B 0,C 180,E1 -4616.035,E2 -4616.035} C_VEL
LIN {X 0,Y 524.755,Z 373.54,A -85,B 0,C 180,E1 -4616.872,E2 -4616.872} C_VEL
LIN {X 0,Y 525.042,Z 361.953,A -85,B 0,C 180,E1 -4617.556,E2 -4617.556} C_VEL
LIN {X 0,Y 525.256,Z 349.271,A -85,B 0,C 180,E1 -4618.118,E2 -4618.118} C_VEL
LIN {X 0,Y 525.444,Z 336.108,A -85,B 0,C 180,E1 -4618.528,E2 -4618.528} C_VEL
LIN {X 0,Y 525.544,Z 322.542,A -85,B 0,C 180,E1 -4618.777,E2 -4618.777} C_VEL
LIN {X 0,Y 525.956,Z 233.28,A -85,B 0,C 180,E1 -4620.003,E2 -4620.003} C_VEL
LIN {X 0,Y 524.223,Z 223.874,A -85,B 0,C 180,E1 -4620.195,E2 -4620.195} C_VEL
LIN {X 0,Y 524.379,Z 209.558,A -85,B 0,C 180,E1 -4622.873,E2 -4622.873} C_VEL
LIN {X 0,Y 524.049,Z 204.5,A -85,B 0,C 180,E1 -4623.829,E2 -4623.829} C_VEL
LIN {X 0,Y 523.988,Z 204.218,A -85,B 0,C 180,E1 -4623.984,E2 -4623.984} C_VEL
LIN {X 0,Y 523.902,Z 204.223,A -85,B 0,C 180,E1 -4627.13,E2 -4627.13} C_VEL
LIN {X 0,Y 523.956,Z 204.222,A -85,B 0,C 180,E1 -4630.132,E2 -4630.132} C_VEL
LIN {X 0,Y 523.93,Z 204.226,A -85,B 0,C 180,E1 -4632.459,E2 -4632.459} C_VEL
LIN {X 0,Y 523.939,Z 204.218,A -85,B 0,C 180,E1 -4635.307,E2 -4635.307} C_VEL
LIN {X 0,Y 523.954,Z 204.217,A -85,B 0,C 180,E1 -4638.686,E2 -4638.686} C_VEL
LIN {X 0,Y 523.905,Z 204.221,A -85,B 0,C 180,E1 -4641.078,E2 -4641.078} C_VEL
LIN {X 0,Y 523.906,Z 204.226,A -85,B 0,C 180,E1 -4643.826,E2 -4643.826} C_VEL
LIN {X 0,Y 523.92,Z 204.22,A -85,B 0,C 180,E1 -4646.634,E2 -4646.634} C_VEL
LIN {X 0,Y 523.938,Z 204.217,A -85,B 0,C 180,E1 -4649.355,E2 -4649.355} C_VEL
LIN {X 0,Y 523.954,Z 204.217,A -85,B 0,C 180,E1 -4652.279,E2 -4652.279} C_VEL
LIN {X 0,Y 523.928,Z 204.216,A -85,B 0,C 180,E1 -4654.58,E2 -4654.58} C_VEL
LIN {X 0,Y 523.93,Z 204.218,A -85,B 0,C 180,E1 -4657.108,E2 -4657.108} C_VEL
LIN {X 0,Y 523.949,Z 204.221,A -85,B 0,C 180,E1 -4659.865,E2 -4659.865} C_VEL
LIN {X 0,Y 523.967,Z 204.211,A -85,B 0,C 180,E1 -4662.837,E2 -4662.837} C_VEL
LIN {X 0,Y 523.972,Z 204.216,A -85,B 0,C 180,E1 -4665.236,E2 -4665.236} C_VEL
LIN {X 0,Y 523.979,Z 204.21,A -85,B 0,C 180,E1 -4668.394,E2 -4668.394} C_VEL
LIN {X 0,Y 523.975,Z 204.216,A -85,B 0,C 180,E1 -4671.516,E2 -4671.516} C_VEL
LIN {X 0,Y 524.016,Z 204.209,A -85,B 0,C 180,E1 -4673.841,E2 -4673.841} C_VEL
LIN {X 0,Y 524.043,Z 204.203,A -85,B 0,C 180,E1 -4676.925,E2 -4676.925} C_VEL
LIN {X 0,Y 524.072,Z 204.198,A -85,B 0,C 180,E1 -4680,E2 -4680} C_VEL
LIN {X 0,Y 524.041,Z 204.208,A -85,B 0,C 180,E1 -4683.075,E2 -4683.075} C_VEL
LIN {X 0,Y 524.002,Z 204.204,A -85,B 0,C 180,E1 -4686.16,E2 -4686.16} C_VEL
LIN {X 0,Y 523.964,Z 204.215,A -85,B 0,C 180,E1 -4689.263,E2 -4689.263} C_VEL
LIN {X 0,Y 523.993,Z 204.208,A -85,B 0,C 180,E1 -4691.752,E2 -4691.752} C_VEL
LIN {X 0,Y 523.96,Z 204.219,A -85,B 0,C 180,E1 -4695.053,E2 -4695.053} C_VEL
LIN {X 0,Y 523.916,Z 204.218,A -85,B 0,C 180,E1 -4697.971,E2 -4697.971} C_VEL
LIN {X 0,Y 523.942,Z 204.218,A -85,B 0,C 180,E1 -4700.412,E2 -4700.412} C_VEL
LIN {X 0,Y 523.878,Z 204.229,A -85,B 0,C 180,E1 -4702.895,E2 -4702.895} C_VEL
LIN {X 0,Y 523.873,Z 204.225,A -85,B 0,C 180,E1 -4705.423,E2 -4705.423} C_VEL
LIN {X 0,Y 523.891,Z 204.222,A -85,B 0,C 180,E1 -4708.004,E2 -4708.004} C_VEL
LIN {X 0,Y 523.913,Z 204.223,A -85,B 0,C 180,E1 -4710.855,E2 -4710.855} C_VEL
LIN {X 0,Y 523.906,Z 204.22,A -85,B 0,C 180,E1 -4713.731,E2 -4713.731} C_VEL
LIN {X 0,Y 523.877,Z 204.232,A -85,B 0,C 180,E1 -4716.402,E2 -4716.402} C_VEL
LIN {X 0,Y 523.893,Z 204.223,A -85,B 0,C 180,E1 -4719.088,E2 -4719.088} C_VEL
LIN {X 0,Y 523.937,Z 204.218,A -85,B 0,C 180,E1 -4722.121,E2 -4722.121} C_VEL
LIN {X 0,Y 523.928,Z 204.217,A -85,B 0,C 180,E1 -4725.312,E2 -4725.312} C_VEL
LIN {X 0,Y 523.927,Z 204.22,A -85,B 0,C 180,E1 -4728.694,E2 -4728.694} C_VEL
LIN {X 0,Y 523.904,Z 204.227,A -85,B 0,C 180,E1 -4731.9,E2 -4731.9} C_VEL
LIN {X 0,Y 523.921,Z 204.22,A -85,B 0,C 180,E1 -4734.912,E2 -4734.912} C_VEL
LIN {X 0,Y 523.93,Z 204.223,A -85,B 0,C 180,E1 -4737.681,E2 -4737.681} C_VEL
LIN {X 0,Y 523.949,Z 204.217,A -85,B 0,C 180,E1 -4740.678,E2 -4740.678} C_VEL
LIN {X 0,Y 523.935,Z 204.224,A -85,B 0,C 180,E1 -4743.728,E2 -4743.728} C_VEL
LIN {X 0,Y 524.018,Z 204.401,A -85,B 0,C 180,E1 -4745.116,E2 -4745.116} C_VEL
LIN {X 0,Y 525.361,Z 211.961,A -85,B 0,C 180,E1 -4746.34,E2 -4746.34} C_VEL
LIN {X 0,Y 525.132,Z 226.936,A -85,B 0,C 180,E1 -4748.612,E2 -4748.612} C_VEL
LIN {X 0,Y 524.602,Z 250.021,A -85,B 0,C 180,E1 -4752.054,E2 -4752.054} C_VEL
LIN {X 0,Y 524.261,Z 269.049,A -85,B 0,C 180,E1 -4754.841,E2 -4754.841} C_VEL
LIN {X 0,Y 525.921,Z 280.515,A -85,B 0,C 180,E1 -4755.048,E2 -4755.048} C_VEL
LIN {X 0,Y 525.489,Z 377.331,A -85,B 0,C 180,E1 -4756.39,E2 -4756.39} C_VEL
LIN {X 0,Y 525.27,Z 390.695,A -85,B 0,C 180,E1 -4756.729,E2 -4756.729} C_VEL
LIN {X 0,Y 524.988,Z 404.045,A -85,B 0,C 180,E1 -4757.239,E2 -4757.239} C_VEL
LIN {X 0,Y 524.754,Z 416.09,A -85,B 0,C 180,E1 -4757.874,E2 -4757.874} C_VEL
LIN {X 0,Y 524.447,Z 428.195,A -85,B 0,C 180,E1 -4758.697,E2 -4758.697} C_VEL
LIN {X 0,Y 524.151,Z 438.433,A -85,B 0,C 180,E1 -4759.571,E2 -4759.571} C_VEL
LIN {X 0,Y 523.917,Z 447.646,A -85,B 0,C 180,E1 -4760.541,E2 -4760.541} C_VEL
LIN {X 0,Y 523.721,Z 456.627,A -85,B 0,C 180,E1 -4761.705,E2 -4761.705} C_VEL
LIN {X 0,Y 523.571,Z 463.857,A -85,B 0,C 180,E1 -4762.867,E2 -4762.867} C_VEL
LIN {X 0,Y 523.487,Z 470.444,A -85,B 0,C 180,E1 -4764.22,E2 -4764.22} C_VEL
LIN {X 0,Y 523.357,Z 474.799,A -85,B 0,C 180,E1 -4765.378,E2 -4765.378} C_VEL
LIN {X 0,Y 523.444,Z 477.112,A -85,B 0,C 180,E1 -4766.15,E2 -4766.15} C_VEL
LIN {X 0,Y 523.368,Z 478.98,A -85,B 0,C 180,E1 -4766.92,E2 -4766.92} C_VEL
LIN {X 0,Y 523.335,Z 480.383,A -85,B 0,C 180,E1 -4767.69,E2 -4767.69} C_VEL
LIN {X 0,Y 523.257,Z 481.994,A -85,B 0,C 180,E1 -4769.229,E2 -4769.229} C_VEL
LIN {X 0,Y 523.259,Z 482.213,A -85,B 0,C 180,E1 -4769.999,E2 -4769.999} C_VEL
LIN {X 0,Y 523.275,Z 481.391,A -85,B 0,C 180,E1 -4771.538,E2 -4771.538} C_VEL
LIN {X 0,Y 523.335,Z 480.397,A -85,B 0,C 180,E1 -4772.307,E2 -4772.307} C_VEL
LIN {X 0,Y 523.367,Z 478.999,A -85,B 0,C 180,E1 -4773.077,E2 -4773.077} C_VEL
LIN {X 0,Y 523.423,Z 476.057,A -85,B 0,C 180,E1 -4774.233,E2 -4774.233} C_VEL
LIN {X 0,Y 523.456,Z 472.071,A -85,B 0,C 180,E1 -4775.391,E2 -4775.391} C_VEL
LIN {X 0,Y 523.496,Z 465.988,A -85,B 0,C 180,E1 -4776.735,E2 -4776.735} C_VEL
LIN {X 0,Y 523.659,Z 459.244,A -85,B 0,C 180,E1 -4777.905,E2 -4777.905} C_VEL
LIN {X 0,Y 523.829,Z 450.936,A -85,B 0,C 180,E1 -4779.068,E2 -4779.068} C_VEL
